LIN {X 0,Y 283.357,Z 583.66,A -85,B 0,C 180,E1 -18703.982,E2 -18703.982} C_VEL
LIN {X 0,Y 286.547,Z 569.765,A -85,B 0,C 180,E1 -18705.445,E2 -18705.445} C_VEL
LIN {X 0,Y 289.347,Z 555.188,A -85,B 0,C 180,E1 -18706.638,E2 -18706.638} C_VEL
LIN {X 0,Y 291.539,Z 540.137,A -85,B 0,C 180,E1 -18707.591,E2 -18707.591} C_VEL
LIN {X 0,Y 293.23,Z 524.888,A -85,B 0,C 180,E1 -18708.256,E2 -18708.256} C_VEL
LIN {X 0,Y 296.275,Z 478.654,A -85,B 0,C 180,E1 -18709.558,E2 -18709.558} C_VEL
LIN {X 0,Y 296.193,Z 472.889,A -85,B 0,C 180,E1 -18709.814,E2 -18709.814} C_VEL
LIN {X 0,Y 293.661,Z 454.463,A -85,B 0,C 180,E1 -18711.157,E2 -18711.157} C_VEL
LIN {X 0,Y 293.71,Z 448.696,A -85,B 0,C 180,E1 -18711.397,E2 -18711.397} C_VEL
LIN {X 0,Y 294.781,Z 433.314,A -85,B 0,C 180,E1 -18711.829,E2 -18711.829} C_VEL
LIN {X 0,Y 289.222,Z 422.71,A -85,B 0,C 180,E1 -18713.709,E2 -18713.709} C_VEL
LIN {X 0,Y 282.657,Z 411.761,A -85,B 0,C 180,E1 -18716.152,E2 -18716.152} C_VEL
LIN {X 0,Y 278.421,Z 405.383,A -85,B 0,C 180,E1 -18717.909,E2 -18717.909} C_VEL
LIN {X 0,Y 275.274,Z 400.843,A -85,B 0,C 180,E1 -18719.325,E2 -18719.325} C_VEL
LIN {X 0,Y 271.812,Z 395.922,A -85,B 0,C 180,E1 -18721.054,E2 -18721.054} C_VEL
LIN {X 0,Y 269.124,Z 392.173,A -85,B 0,C 180,E1 -18722.549,E2 -18722.549} C_VEL
LIN {X 0,Y 265.588,Z 388.374,A -85,B 0,C 180,E1 -18724.695,E2 -18724.695} C_VEL
LIN {X 0,Y 264.483,Z 386.612,A -85,B 0,C 180,E1 -18725.479,E2 -18725.479} C_VEL
LIN {X 0,Y 261.658,Z 384.021,A -85,B 0,C 180,E1 -18727.62,E2 -18727.62} C_VEL
LIN {X 0,Y 260.222,Z 381.079,A -85,B 0,C 180,E1 -18729.082,E2 -18729.082} C_VEL
LIN {X 0,Y 256.877,Z 379.067,A -85,B 0,C 180,E1 -18732.843,E2 -18732.843} C_VEL
LIN {X 0,Y 255.223,Z 375.845,A -85,B 0,C 180,E1 -18737.016,E2 -18737.016} C_VEL
LIN {X 0,Y 254.832,Z 376.279,A -85,B 0,C 180,E1 -18740.587,E2 -18740.587} C_VEL
LIN {X 0,Y 256.37,Z 378.534,A -85,B 0,C 180,E1 -18745.48,E2 -18745.48} C_VEL
LIN {X 0,Y 260.204,Z 384.567,A -85,B 0,C 180,E1 -18750.484,E2 -18750.484} C_VEL
LIN {X 0,Y 262.637,Z 387.768,A -85,B 0,C 180,E1 -18752.64,E2 -18752.64} C_VEL
LIN {X 0,Y 267.7,Z 395.205,A -85,B 0,C 180,E1 -18756.153,E2 -18756.153} C_VEL
LIN {X 0,Y 272.191,Z 402.334,A -85,B 0,C 180,E1 -18758.706,E2 -18758.706} C_VEL
LIN {X 0,Y 275.6,Z 407.992,A -85,B 0,C 180,E1 -18760.404,E2 -18760.404} C_VEL
LIN {X 0,Y 279.037,Z 414.108,A -85,B 0,C 180,E1 -18761.968,E2 -18761.968} C_VEL
LIN {X 0,Y 282.488,Z 420.477,A -85,B 0,C 180,E1 -18763.419,E2 -18763.419} C_VEL
LIN {X 0,Y 286.498,Z 428.65,A -85,B 0,C 180,E1 -18764.998,E2 -18764.998} C_VEL
LIN {X 0,Y 291.285,Z 439.57,A -85,B 0,C 180,E1 -18766.767,E2 -18766.767} C_VEL
LIN {X 0,Y 293.256,Z 444.964,A -85,B 0,C 180,E1 -18767.491,E2 -18767.491} C_VEL
LIN {X 0,Y 293.808,Z 453.087,A -85,B 0,C 180,E1 -18767.982,E2 -18767.982} C_VEL
LIN {X 0,Y 287.202,Z 546.54,A -85,B 0,C 180,E1 -18770.544,E2 -18770.544} C_VEL
LIN {X 0,Y 285.082,Z 562.821,A -85,B 0,C 180,E1 -18771.219,E2 -18771.219} C_VEL
LIN {X 0,Y 282.431,Z 577.753,A -85,B 0,C 180,E1 -18772.097,E2 -18772.097} C_VEL
LIN {X 0,Y 279.427,Z 591.001,A -85,B 0,C 180,E1 -18773.094,E2 -18773.094} C_VEL
LIN {X 0,Y 275.993,Z 604.177,A -85,B 0,C 180,E1 -18774.373,E2 -18774.373} C_VEL
LIN {X 0,Y 271.998,Z 617.923,A -85,B 0,C 180,E1 -18776.047,E2 -18776.047} C_VEL
LIN {X 0,Y 268.029,Z 630.286,A -85,B 0,C 180,E1 -18777.928,E2 -18777.928} C_VEL
LIN {X 0,Y 263.932,Z 641.731,A -85,B 0,C 180,E1 -18780.047,E2 -18780.047} C_VEL
LIN {X 0,Y 260.339,Z 651.436,A -85,B 0,C 180,E1 -18782.245,E2 -18782.245} C_VEL
LIN {X 0,Y 256.679,Z 661.36,A -85,B 0,C 180,E1 -18784.988,E2 -18784.988} C_VEL
LIN {X 0,Y 253.789,Z 669.171,A -85,B 0,C 180,E1 -18787.618,E2 -18787.618} C_VEL
LIN {X 0,Y 251.343,Z 675.969,A -85,B 0,C 180,E1 -18790.394,E2 -18790.394} C_VEL
LIN {X 0,Y 249.28,Z 682.278,A -85,B 0,C 180,E1 -18793.624,E2 -18793.624} C_VEL
LIN {X 0,Y 247.949,Z 687.204,A -85,B 0,C 180,E1 -18796.893,E2 -18796.893} C_VEL
LIN {X 0,Y 247.209,Z 690.852,A -85,B 0,C 180,E1 -18800.178,E2 -18800.178} C_VEL
LIN {X 0,Y 247.023,Z 693.292,A -85,B 0,C 180,E1 -18803.465,E2 -18803.465} C_VEL
LIN {X 0,Y 247.109,Z 694.554,A -85,B 0,C 180,E1 -18806.738,E2 -18806.738} C_VEL
LIN {X 0,Y 247.232,Z 694.628,A -85,B 0,C 180,E1 -18809.999,E2 -18809.999} C_VEL
LIN {X 0,Y 247.155,Z 693.435,A -85,B 0,C 180,E1 -18813.26,E2 -18813.26} C_VEL
LIN {X 0,Y 247.05,Z 690.958,A -85,B 0,C 180,E1 -18816.533,E2 -18816.533} C_VEL
LIN {X 0,Y 247.256,Z 687.184,A -85,B 0,C 180,E1 -18819.819,E2 -18819.819} C_VEL
LIN {X 0,Y 247.912,Z 682.014,A -85,B 0,C 180,E1 -18823.107,E2 -18823.107} C_VEL
LIN {X 0,Y 249.216,Z 675.046,A -85,B 0,C 180,E1 -18826.503,E2 -18826.503} C_VEL
LIN {X 0,Y 250.99,Z 666.908,A -85,B 0,C 180,E1 -18829.633,E2 -18829.633} C_VEL
LIN {X 0,Y 253.326,Z 657.918,A -85,B 0,C 180,E1 -18832.424,E2 -18832.424} C_VEL
LIN {X 0,Y 255.53,Z 648.604,A -85,B 0,C 180,E1 -18834.823,E2 -18834.823} C_VEL
LIN {X 0,Y 258.296,Z 637.846,A -85,B 0,C 180,E1 -18837.112,E2 -18837.112} C_VEL
LIN {X 0,Y 261.218,Z 626.014,A -85,B 0,C 180,E1 -18839.185,E2 -18839.185} C_VEL
LIN {X 0,Y 264.274,Z 613.144,A -85,B 0,C 180,E1 -18841.013,E2 -18841.013} C_VEL
LIN {X 0,Y 266.977,Z 600.152,A -85,B 0,C 180,E1 -18842.513,E2 -18842.513} C_VEL
LIN {X 0,Y 269.556,Z 585.357,A -85,B 0,C 180,E1 -18843.868,E2 -18843.868} C_VEL
LIN {X 0,Y 271.862,Z 570.467,A -85,B 0,C 180,E1 -18844.886,E2 -18844.886} C_VEL
LIN {X 0,Y 273.597,Z 555.142,A -85,B 0,C 180,E1 -18845.646,E2 -18845.646} C_VEL
LIN {X 0,Y 274.669,Z 537.879,A -85,B 0,C 180,E1 -18846.22,E2 -18846.22} C_VEL
LIN {X 0,Y 279.129,Z 449.321,A -85,B 0,C 180,E1 -18848.643,E2 -18848.643} C_VEL
LIN {X 0,Y 276.743,Z 432.647,A -85,B 0,C 180,E1 -18849.535,E2 -18849.535} C_VEL
LIN {X 0,Y 270.603,Z 418.098,A -85,B 0,C 180,E1 -18850.922,E2 -18850.922} C_VEL
LIN {X 0,Y 262.703,Z 401.029,A -85,B 0,C 180,E1 -18852.765,E2 -18852.765} C_VEL
LIN {X 0,Y 254.764,Z 385.449,A -85,B 0,C 180,E1 -18854.695,E2 -18854.695} C_VEL
LIN {X 0,Y 252.687,Z 381.306,A -85,B 0,C 180,E1 -18855.25,E2 -18855.25} C_VEL
LIN {X 0,Y 249.885,Z 372.112,A -85,B 0,C 180,E1 -18858.629,E2 -18858.629} C_VEL
LIN {X 0,Y 249.014,Z 369.094,A -85,B 0,C 180,E1 -18859.866,E2 -18859.866} C_VEL
LIN {X 0,Y 249.045,Z 369.092,A -85,B 0,C 180,E1 -18863.658,E2 -18863.658} C_VEL
LIN {X 0,Y 249.034,Z 369.085,A -85,B 0,C 180,E1 -18867.846,E2 -18867.846} C_VEL
LIN {X 0,Y 249.094,Z 369.082,A -85,B 0,C 180,E1 -18871.339,E2 -18871.339} C_VEL
LIN {X 0,Y 249.148,Z 369.073,A -85,B 0,C 180,E1 -18874.969,E2 -18874.969} C_VEL
LIN {X 0,Y 249.108,Z 369.08,A -85,B 0,C 180,E1 -18880.212,E2 -18880.212} C_VEL
LIN {X 0,Y 249.239,Z 369.065,A -85,B 0,C 180,E1 -18883.622,E2 -18883.622} C_VEL
LIN {X 0,Y 249.25,Z 369.033,A -85,B 0,C 180,E1 -18888.617,E2 -18888.617} C_VEL
LIN {X 0,Y 249.477,Z 369.026,A -85,B 0,C 180,E1 -18891.903,E2 -18891.903} C_VEL
LIN {X 0,Y 249.434,Z 369.031,A -85,B 0,C 180,E1 -18896.77,E2 -18896.77} C_VEL
LIN {X 0,Y 249.726,Z 368.993,A -85,B 0,C 180,E1 -18900.001,E2 -18900.001} C_VEL
LIN {X 0,Y 249.434,Z 369.038,A -85,B 0,C 180,E1 -18903.231,E2 -18903.231} C_VEL
LIN {X 0,Y 249.482,Z 369.017,A -85,B 0,C 180,E1 -18908.098,E2 -18908.098} C_VEL
LIN {X 0,Y 249.251,Z 369.062,A -85,B 0,C 180,E1 -18911.384,E2 -18911.384} C_VEL
LIN {X 0,Y 249.24,Z 369.043,A -85,B 0,C 180,E1 -18916.379,E2 -18916.379} C_VEL
LIN {X 0,Y 249.083,Z 369.081,A -85,B 0,C 180,E1 -18921.519,E2 -18921.519} C_VEL
LIN {X 0,Y 249.116,Z 369.057,A -85,B 0,C 180,E1 -18925.476,E2 -18925.476} C_VEL
LIN {X 0,Y 249.082,Z 369.082,A -85,B 0,C 180,E1 -18928.994,E2 -18928.994} C_VEL
LIN {X 0,Y 249.03,Z 369.085,A -85,B 0,C 180,E1 -18932.427,E2 -18932.427} C_VEL
LIN {X 0,Y 249.029,Z 369.076,A -85,B 0,C 180,E1 -18936.346,E2 -18936.346} C_VEL
LIN {X 0,Y 249.006,Z 369.092,A -85,B 0,C 180,E1 -18940.479,E2 -18940.479} C_VEL
LIN {X 0,Y 248.986,Z 369.084,A -85,B 0,C 180,E1 -18944.884,E2 -18944.884} C_VEL
LIN {X 0,Y 249.01,Z 369.092,A -85,B 0,C 180,E1 -18947.363,E2 -18947.363} C_VEL
LIN {X 0,Y 249.026,Z 369.075,A -85,B 0,C 180,E1 -18951.62,E2 -18951.62} C_VEL
LIN {X 0,Y 249.045,Z 369.087,A -85,B 0,C 180,E1 -18955.641,E2 -18955.641} C_VEL
LIN {X 0,Y 249.004,Z 369.087,A -85,B 0,C 180,E1 -18959.468,E2 -18959.468} C_VEL
LIN {X 0,Y 249.039,Z 369.082,A -85,B 0,C 180,E1 -18963.159,E2 -18963.159} C_VEL
LIN {X 0,Y 249.059,Z 369.087,A -85,B 0,C 180,E1 -18966.731,E2 -18966.731} C_VEL
LIN {X 0,Y 249.078,Z 369.076,A -85,B 0,C 180,E1 -18970.21,E2 -18970.21} C_VEL
LIN {X 0,Y 249.16,Z 369.069,A -85,B 0,C 180,E1 -18973.617,E2 -18973.617} C_VEL
LIN {X 0,Y 249.23,Z 369.06,A -85,B 0,C 180,E1 -18978.616,E2 -18978.616} C_VEL
LIN {X 0,Y 249.421,Z 369.036,A -85,B 0,C 180,E1 -18981.902,E2 -18981.902} C_VEL
LIN {X 0,Y 249.324,Z 369.179,A -85,B 0,C 180,E1 -18984.744,E2 -18984.744} C_VEL
LIN {X 0,Y 250.266,Z 371.871,A -85,B 0,C 180,E1 -18985.028,E2 -18985.028} C_VEL
LIN {X 0,Y 252.185,Z 374.531,A -85,B 0,C 180,E1 -18985.484,E2 -18985.484} C_VEL
LIN {X 0,Y 259.111,Z 385.318,A -85,B 0,C 180,E1 -18987.119,E2 -18987.119} C_VEL
LIN {X 0,Y 266.091,Z 397.678,A -85,B 0,C 180,E1 -18988.707,E2 -18988.707} C_VEL
LIN {X 0,Y 276.646,Z 417.563,A -85,B 0,C 180,E1 -18990.978,E2 -18990.978} C_VEL
LIN {X 0,Y 279.769,Z 424.265,A -85,B 0,C 180,E1 -18991.636,E2 -18991.636} C_VEL
LIN {X 0,Y 274.746,Z 521.539,A -85,B 0,C 180,E1 -18994.319,E2 -18994.319} C_VEL
LIN {X 0,Y 273.393,Z 537.132,A -85,B 0,C 180,E1 -18995.024,E2 -18995.024} C_VEL
LIN {X 0,Y 271.599,Z 552.606,A -85,B 0,C 180,E1 -18996.035,E2 -18996.035} C_VEL
LIN {X 0,Y 269.275,Z 567.725,A -85,B 0,C 180,E1 -18997.341,E2 -18997.341} C_VEL
LIN {X 0,Y 266.738,Z 581.835,A -85,B 0,C 180,E1 -18998.906,E2 -18998.906} C_VEL
LIN {X 0,Y 263.885,Z 595.218,A -85,B 0,C 180,E1 -19000.745,E2 -19000.745} C_VEL
LIN {X 0,Y 261.136,Z 607.122,A -85,B 0,C 180,E1 -19002.757,E2 -19002.757} C_VEL
LIN {X 0,Y 258.433,Z 617.973,A -85,B 0,C 180,E1 -19004.973,E2 -19004.973} C_VEL
LIN {X 0,Y 255.678,Z 628.541,A -85,B 0,C 180,E1 -19007.6,E2 -19007.6} C_VEL
LIN {X 0,Y 253.251,Z 637.668,A -85,B 0,C 180,E1 -19010.377,E2 -19010.377} C_VEL
LIN {X 0,Y 251.383,Z 644.892,A -85,B 0,C 180,E1 -19013.043,E2 -19013.043} C_VEL
LIN {X 0,Y 249.835,Z 651.011,A -85,B 0,C 180,E1 -19015.817,E2 -19015.817} C_VEL
LIN {X 0,Y 248.671,Z 656.327,A -85,B 0,C 180,E1 -19018.82,E2 -19018.82} C_VEL
LIN {X 0,Y 247.816,Z 660.314,A -85,B 0,C 180,E1 -19021.701,E2 -19021.701} C_VEL
LIN {X 0,Y 247.184,Z 663.356,A -85,B 0,C 180,E1 -19024.657,E2 -19024.657} C_VEL
LIN {X 0,Y 246.893,Z 665.098,A -85,B 0,C 180,E1 -19027.15,E2 -19027.15} C_VEL
LIN {X 0,Y 246.829,Z 666.221,A -85,B 0,C 180,E1 -19029.755,E2 -19029.755} C_VEL
LIN {X 0,Y 247.029,Z 666.573,A -85,B 0,C 180,E1 -19033.064,E2 -19033.064} C_VEL
LIN {X 0,Y 247.33,Z 666.182,A -85,B 0,C 180,E1 -19035.267,E2 -19035.267} C_VEL
LIN {X 0,Y 247.839,Z 665.251,A -85,B 0,C 180,E1 -19037.502,E2 -19037.502} C_VEL
LIN {X 0,Y 248.563,Z 663.696,A -85,B 0,C 180,E1 -19039.767,E2 -19039.767} C_VEL
LIN {X 0,Y 249.902,Z 660.558,A -85,B 0,C 180,E1 -19042.977,E2 -19042.977} C_VEL
LIN {X 0,Y 251.711,Z 656.351,A -85,B 0,C 180,E1 -19046.053,E2 -19046.053} C_VEL
LIN {X 0,Y 254.029,Z 650.936,A -85,B 0,C 180,E1 -19049.055,E2 -19049.055} C_VEL
LIN {X 0,Y 256.731,Z 644.578,A -85,B 0,C 180,E1 -19051.849,E2 -19051.849} C_VEL
LIN {X 0,Y 260.219,Z 636.264,A -85,B 0,C 180,E1 -19054.772,E2 -19054.772} C_VEL
LIN {X 0,Y 263.779,Z 627.473,A -85,B 0,C 180,E1 -19057.274,E2 -19057.274} C_VEL
LIN {X 0,Y 267.474,Z 617.456,A -85,B 0,C 180,E1 -19059.625,E2 -19059.625} C_VEL
LIN {X 0,Y 271.215,Z 606.687,A -85,B 0,C 180,E1 -19061.687,E2 -19061.687} C_VEL
LIN {X 0,Y 274.829,Z 595.249,A -85,B 0,C 180,E1 -19063.488,E2 -19063.488} C_VEL
LIN {X 0,Y 278.429,Z 582.521,A -85,B 0,C 180,E1 -19065.12,E2 -19065.12} C_VEL
LIN {X 0,Y 281.53,Z 569.386,A -85,B 0,C 180,E1 -19066.501,E2 -19066.501} C_VEL
LIN {X 0,Y 284.323,Z 555.435,A -85,B 0,C 180,E1 -19067.644,E2 -19067.644} C_VEL
LIN {X 0,Y 286.501,Z 541.074,A -85,B 0,C 180,E1 -19068.561,E2 -19068.561} C_VEL
LIN {X 0,Y 288.235,Z 525.976,A -85,B 0,C 180,E1 -19069.24,E2 -19069.24} C_VEL
LIN {X 0,Y 291.553,Z 478.481,A -85,B 0,C 180,E1 -19070.59,E2 -19070.59} C_VEL
LIN {X 0,Y 293.71,Z 448.696,A -85,B 0,C 180,E1 -19071.397,E2 -19071.397} C_VEL
LIN {X 0,Y 293.59,Z 444.895,A -85,B 0,C 180,E1 -19071.596,E2 -19071.596} C_VEL
LIN {X 0,Y 292.386,Z 440.371,A -85,B 0,C 180,E1 -19072.09,E2 -19072.09} C_VEL
LIN {X 0,Y 289.941,Z 435.432,A -85,B 0,C 180,E1 -19072.925,E2 -19072.925} C_VEL
LIN {X 0,Y 287.813,Z 431.718,A -85,B 0,C 180,E1 -19073.65,E2 -19073.65} C_VEL
LIN {X 0,Y 282.661,Z 422.453,A -85,B 0,C 180,E1 -19075.585,E2 -19075.585} C_VEL
LIN {X 0,Y 277.736,Z 414.214,A -85,B 0,C 180,E1 -19077.626,E2 -19077.626} C_VEL
LIN {X 0,Y 271.268,Z 404.805,A -85,B 0,C 180,E1 -19080.664,E2 -19080.664} C_VEL
LIN {X 0,Y 269.595,Z 402.252,A -85,B 0,C 180,E1 -19081.563,E2 -19081.563} C_VEL
LIN {X 0,Y 266.623,Z 398.146,A -85,B 0,C 180,E1 -19083.305,E2 -19083.305} C_VEL
LIN {X 0,Y 263.648,Z 394.765,A -85,B 0,C 180,E1 -19085.209,E2 -19085.209} C_VEL
LIN {X 0,Y 262.663,Z 393.245,A -85,B 0,C 180,E1 -19085.951,E2 -19085.951} C_VEL
LIN {X 0,Y 259.912,Z 390.436,A -85,B 0,C 180,E1 -19088.174,E2 -19088.174} C_VEL
LIN {X 0,Y 258.564,Z 387.874,A -85,B 0,C 180,E1 -19089.583,E2 -19089.583} C_VEL
LIN {X 0,Y 255.368,Z 385.663,A -85,B 0,C 180,E1 -19093.528,E2 -19093.528} C_VEL
LIN {X 0,Y 254.133,Z 382.889,A -85,B 0,C 180,E1 -19097.092,E2 -19097.092} C_VEL
LIN {X 0,Y 253.747,Z 383.264,A -85,B 0,C 180,E1 -19100.403,E2 -19100.403} C_VEL
LIN {X 0,Y 255.238,Z 385.561,A -85,B 0,C 180,E1 -19105.397,E2 -19105.397} C_VEL
LIN {X 0,Y 258.718,Z 391.354,A -85,B 0,C 180,E1 -19110.142,E2 -19110.142} C_VEL
LIN {X 0,Y 260.948,Z 394.357,A -85,B 0,C 180,E1 -19112.188,E2 -19112.188} C_VEL
LIN {X 0,Y 265.509,Z 401.376,A -85,B 0,C 180,E1 -19115.551,E2 -19115.551} C_VEL
LIN {X 0,Y 269.578,Z 408.07,A -85,B 0,C 180,E1 -19118.001,E2 -19118.001} C_VEL
LIN {X 0,Y 273.017,Z 414.016,A -85,B 0,C 180,E1 -19119.814,E2 -19119.814} C_VEL
LIN {X 0,Y 275.844,Z 419.193,A -85,B 0,C 180,E1 -19121.173,E2 -19121.173} C_VEL
LIN {X 0,Y 280.027,Z 427.177,A -85,B 0,C 180,E1 -19123.026,E2 -19123.026} C_VEL
LIN {X 0,Y 284.416,Z 436.813,A -85,B 0,C 180,E1 -19124.823,E2 -19124.823} C_VEL
LIN {X 0,Y 288.38,Z 446.669,A -85,B 0,C 180,E1 -19126.365,E2 -19126.365} C_VEL
LIN {X 0,Y 288.92,Z 448.494,A -85,B 0,C 180,E1 -19126.586,E2 -19126.586} C_VEL
LIN {X 0,Y 289.262,Z 453.9,A -85,B 0,C 180,E1 -19126.92,E2 -19126.92} C_VEL
LIN {X 0,Y 282.349,Z 546.363,A -85,B 0,C 180,E1 -19129.495,E2 -19129.495} C_VEL
LIN {X 0,Y 280.173,Z 562.533,A -85,B 0,C 180,E1 -19130.175,E2 -19130.175} C_VEL
LIN {X 0,Y 277.653,Z 576.328,A -85,B 0,C 180,E1 -19130.976,E2 -19130.976} C_VEL
LIN {X 0,Y 274.318,Z 590.651,A -85,B 0,C 180,E1 -19132.056,E2 -19132.056} C_VEL
LIN {X 0,Y 270.342,Z 605.304,A -85,B 0,C 180,E1 -19133.51,E2 -19133.51} C_VEL
LIN {X 0,Y 266.188,Z 618.701,A -85,B 0,C 180,E1 -19135.201,E2 -19135.201} C_VEL
LIN {X 0,Y 262.061,Z 630.826,A -85,B 0,C 180,E1 -19137.106,E2 -19137.106} C_VEL
LIN {X 0,Y 257.817,Z 642.124,A -85,B 0,C 180,E1 -19139.261,E2 -19139.261} C_VEL
LIN {X 0,Y 253.476,Z 653.199,A -85,B 0,C 180,E1 -19141.877,E2 -19141.877} C_VEL
LIN {X 0,Y 250.028,Z 661.958,A -85,B 0,C 180,E1 -19144.443,E2 -19144.443} C_VEL
LIN {X 0,Y 247.197,Z 669.166,A -85,B 0,C 180,E1 -19146.987,E2 -19146.987} C_VEL
LIN {X 0,Y 244.593,Z 675.876,A -85,B 0,C 180,E1 -19149.83,E2 -19149.83} C_VEL
LIN {X 0,Y 242.422,Z 682.119,A -85,B 0,C 180,E1 -19153.147,E2 -19153.147} C_VEL
LIN {X 0,Y 240.967,Z 686.994,A -85,B 0,C 180,E1 -19156.506,E2 -19156.506} C_VEL
LIN {X 0,Y 240.139,Z 690.566,A -85,B 0,C 180,E1 -19159.886,E2 -19159.886} C_VEL
LIN {X 0,Y 239.941,Z 692.948,A -85,B 0,C 180,E1 -19163.271,E2 -19163.271} C_VEL
LIN {X 0,Y 240.018,Z 694.15,A -85,B 0,C 180,E1 -19166.642,E2 -19166.642} C_VEL
LIN {X 0,Y 240.152,Z 694.166,A -85,B 0,C 180,E1 -19169.999,E2 -19169.999} C_VEL
LIN {X 0,Y 240.061,Z 692.937,A -85,B 0,C 180,E1 -19173.356,E2 -19173.356} C_VEL
LIN {X 0,Y 239.965,Z 690.401,A -85,B 0,C 180,E1 -19176.727,E2 -19176.727} C_VEL
LIN {X 0,Y 240.197,Z 686.556,A -85,B 0,C 180,E1 -19180.11,E2 -19180.11} C_VEL
LIN {X 0,Y 240.917,Z 681.31,A -85,B 0,C 180,E1 -19183.495,E2 -19183.495} C_VEL
LIN {X 0,Y 242.259,Z 674.532,A -85,B 0,C 180,E1 -19186.863,E2 -19186.863} C_VEL
LIN {X 0,Y 243.917,Z 667.174,A -85,B 0,C 180,E1 -19189.788,E2 -19189.788} C_VEL
LIN {X 0,Y 246.293,Z 658.32,A -85,B 0,C 180,E1 -19192.657,E2 -19192.657} C_VEL
LIN {X 0,Y 248.949,Z 647.763,A -85,B 0,C 180,E1 -19195.454,E2 -19195.454} C_VEL
LIN {X 0,Y 251.88,Z 636.593,A -85,B 0,C 180,E1 -19197.862,E2 -19197.862} C_VEL
LIN {X 0,Y 254.953,Z 624.595,A -85,B 0,C 180,E1 -19199.975,E2 -19199.975} C_VEL
LIN {X 0,Y 258.076,Z 611.495,A -85,B 0,C 180,E1 -19201.844,E2 -19201.844} C_VEL
LIN {X 0,Y 261.12,Z 597.349,A -85,B 0,C 180,E1 -19203.451,E2 -19203.451} C_VEL
LIN {X 0,Y 263.641,Z 583.048,A -85,B 0,C 180,E1 -19204.736,E2 -19204.736} C_VEL
LIN {X 0,Y 265.994,Z 567.521,A -85,B 0,C 180,E1 -19205.772,E2 -19205.772} C_VEL
LIN {X 0,Y 267.644,Z 552.107,A -85,B 0,C 180,E1 -19206.506,E2 -19206.506} C_VEL
LIN {X 0,Y 269.042,Z 528.766,A -85,B 0,C 180,E1 -19207.22,E2 -19207.22} C_VEL
LIN {X 0,Y 273.126,Z 450.076,A -85,B 0,C 180,E1 -19209.419,E2 -19209.419} C_VEL
LIN {X 0,Y 271.018,Z 435.37,A -85,B 0,C 180,E1 -19210.238,E2 -19210.238} C_VEL
LIN {X 0,Y 263.905,Z 418.352,A -85,B 0,C 180,E1 -19211.925,E2 -19211.925} C_VEL
LIN {X 0,Y 254.711,Z 398.936,A -85,B 0,C 180,E1 -19214.161,E2 -19214.161} C_VEL
LIN {X 0,Y 247.112,Z 384.535,A -85,B 0,C 180,E1 -19216.104,E2 -19216.104} C_VEL
LIN {X 0,Y 245.235,Z 380.665,A -85,B 0,C 180,E1 -19216.686,E2 -19216.686} C_VEL
LIN {X 0,Y 241.99,Z 369.959,A -85,B 0,C 180,E1 -19220.853,E2 -19220.853} C_VEL
LIN {X 0,Y 241.985,Z 369.974,A -85,B 0,C 180,E1 -19224.489,E2 -19224.489} C_VEL
LIN {X 0,Y 241.972,Z 369.97,A -85,B 0,C 180,E1 -19228.48,E2 -19228.48} C_VEL
LIN {X 0,Y 242.006,Z 369.966,A -85,B 0,C 180,E1 -19232.313,E2 -19232.313} C_VEL
LIN {X 0,Y 242.054,Z 369.958,A -85,B 0,C 180,E1 -19236.016,E2 -19236.016} C_VEL
LIN {X 0,Y 242.035,Z 369.962,A -85,B 0,C 180,E1 -19239.608,E2 -19239.608} C_VEL
LIN {X 0,Y 242.16,Z 369.947,A -85,B 0,C 180,E1 -19243.279,E2 -19243.279} C_VEL
LIN {X 0,Y 242.184,Z 369.913,A -85,B 0,C 180,E1 -19248.28,E2 -19248.28} C_VEL
LIN {X 0,Y 242.424,Z 369.9,A -85,B 0,C 180,E1 -19251.666,E2 -19251.666} C_VEL
LIN {X 0,Y 242.257,Z 369.934,A -85,B 0,C 180,E1 -19255.008,E2 -19255.008} C_VEL
LIN {X 0,Y 242.634,Z 369.868,A -85,B 0,C 180,E1 -19258.341,E2 -19258.341} C_VEL
LIN {X 0,Y 242.635,Z 369.884,A -85,B 0,C 180,E1 -19261.66,E2 -19261.66} C_VEL
LIN {X 0,Y 242.429,Z 369.893,A -85,B 0,C 180,E1 -19266.709,E2 -19266.709} C_VEL
LIN {X 0,Y 242.344,Z 369.917,A -85,B 0,C 180,E1 -19270.021,E2 -19270.021} C_VEL
LIN {X 0,Y 242.165,Z 369.928,A -85,B 0,C 180,E1 -19275.142,E2 -19275.142} C_VEL
LIN {X 0,Y 242.071,Z 369.947,A -85,B 0,C 180,E1 -19278.625,E2 -19278.625} C_VEL
LIN {X 0,Y 242.005,Z 369.964,A -85,B 0,C 180,E1 -19282.181,E2 -19282.181} C_VEL
LIN {X 0,Y 242.065,Z 369.933,A -85,B 0,C 180,E1 -19285.839,E2 -19285.839} C_VEL
LIN {X 0,Y 242.029,Z 369.96,A -85,B 0,C 180,E1 -19289.581,E2 -19289.581} C_VEL
LIN {X 0,Y 241.98,Z 369.956,A -85,B 0,C 180,E1 -19293.494,E2 -19293.494} C_VEL
LIN {X 0,Y 241.986,Z 369.962,A -85,B 0,C 180,E1 -19297.583,E2 -19297.583} C_VEL
LIN {X 0,Y 241.933,Z 369.965,A -85,B 0,C 180,E1 -19301.924,E2 -19301.924} C_VEL
LIN {X 0,Y 241.926,Z 369.974,A -85,B 0,C 180,E1 -19306.575,E2 -19306.575} C_VEL
LIN {X 0,Y 241.957,Z 369.959,A -85,B 0,C 180,E1 -19310.282,E2 -19310.282} C_VEL
LIN {X 0,Y 241.989,Z 369.969,A -85,B 0,C 180,E1 -19314.49,E2 -19314.49} C_VEL
LIN {X 0,Y 241.954,Z 369.959,A -85,B 0,C 180,E1 -19318.478,E2 -19318.478} C_VEL
LIN {X 0,Y 241.972,Z 369.968,A -85,B 0,C 180,E1 -19322.309,E2 -19322.309} C_VEL
LIN {X 0,Y 242.029,Z 369.958,A -85,B 0,C 180,E1 -19326.014,E2 -19326.014} C_VEL
LIN {X 0,Y 242.018,Z 369.953,A -85,B 0,C 180,E1 -19329.607,E2 -19329.607} C_VEL
LIN {X 0,Y 242.108,Z 369.948,A -85,B 0,C 180,E1 -19333.325,E2 -19333.325} C_VEL
LIN {X 0,Y 242.162,Z 369.939,A -85,B 0,C 180,E1 -19338.279,E2 -19338.279} C_VEL
LIN {X 0,Y 242.375,Z 369.913,A -85,B 0,C 180,E1 -19341.665,E2 -19341.665} C_VEL
LIN {X 0,Y 242.394,Z 369.918,A -85,B 0,C 180,E1 -19343.435,E2 -19343.435} C_VEL
LIN {X 0,Y 243.474,Z 372.961,A -85,B 0,C 180,E1 -19343.802,E2 -19343.802} C_VEL
LIN {X 0,Y 245.055,Z 375.31,A -85,B 0,C 180,E1 -19344.207,E2 -19344.207} C_VEL
LIN {X 0,Y 254.562,Z 390.102,A -85,B 0,C 180,E1 -19346.535,E2 -19346.535} C_VEL
LIN {X 0,Y 261.4,Z 402.403,A -85,B 0,C 180,E1 -19348.153,E2 -19348.153} C_VEL
LIN {X 0,Y 271.387,Z 421.335,A -85,B 0,C 180,E1 -19350.363,E2 -19350.363} C_VEL
LIN {X 0,Y 273.748,Z 426.672,A -85,B 0,C 180,E1 -19350.889,E2 -19350.889} C_VEL
LIN {X 0,Y 268.582,Z 522.332,A -85,B 0,C 180,E1 -19353.583,E2 -19353.583} C_VEL
LIN {X 0,Y 267.21,Z 537.779,A -85,B 0,C 180,E1 -19354.303,E2 -19354.303} C_VEL
LIN {X 0,Y 265.385,Z 553.005,A -85,B 0,C 180,E1 -19355.319,E2 -19355.319} C_VEL
LIN {X 0,Y 263.047,Z 567.686,A -85,B 0,C 180,E1 -19356.603,E2 -19356.603} C_VEL
LIN {X 0,Y 260.519,Z 581.439,A -85,B 0,C 180,E1 -19358.143,E2 -19358.143} C_VEL
LIN {X 0,Y 257.633,Z 594.717,A -85,B 0,C 180,E1 -19359.982,E2 -19359.982} C_VEL
LIN {X 0,Y 254.863,Z 606.282,A -85,B 0,C 180,E1 -19361.937,E2 -19361.937} C_VEL
LIN {X 0,Y 252.003,Z 617.513,A -85,B 0,C 180,E1 -19364.244,E2 -19364.244} C_VEL
LIN {X 0,Y 249.11,Z 628.183,A -85,B 0,C 180,E1 -19366.917,E2 -19366.917} C_VEL
LIN {X 0,Y 246.515,Z 637.583,A -85,B 0,C 180,E1 -19369.81,E2 -19369.81} C_VEL
LIN {X 0,Y 244.275,Z 645.879,A -85,B 0,C 180,E1 -19372.974,E2 -19372.974} C_VEL
LIN {X 0,Y 242.609,Z 652.448,A -85,B 0,C 180,E1 -19376.099,E2 -19376.099} C_VEL
LIN {X 0,Y 241.452,Z 657.514,A -85,B 0,C 180,E1 -19379.164,E2 -19379.164} C_VEL
LIN {X 0,Y 240.613,Z 661.264,A -85,B 0,C 180,E1 -19382.106,E2 -19382.106} C_VEL
LIN {X 0,Y 239.903,Z 664.66,A -85,B 0,C 180,E1 -19385.868,E2 -19385.868} C_VEL
LIN {X 0,Y 239.749,Z 665.917,A -85,B 0,C 180,E1 -19387.996,E2 -19387.996} C_VEL
LIN {X 0,Y 239.753,Z 666.78,A -85,B 0,C 180,E1 -19390.345,E2 -19390.345} C_VEL
LIN {X 0,Y 239.923,Z 667.017,A -85,B 0,C 180,E1 -19392.918,E2 -19392.918} C_VEL
LIN {X 0,Y 240.276,Z 666.651,A -85,B 0,C 180,E1 -19395.412,E2 -19395.412} C_VEL
LIN {X 0,Y 240.846,Z 665.711,A -85,B 0,C 180,E1 -19397.843,E2 -19397.843} C_VEL
LIN {X 0,Y 242.198,Z 663.013,A -85,B 0,C 180,E1 -19401.581,E2 -19401.581} C_VEL
LIN {X 0,Y 243.836,Z 659.445,A -85,B 0,C 180,E1 -19404.798,E2 -19404.798} C_VEL
LIN {X 0,Y 245.991,Z 654.689,A -85,B 0,C 180,E1 -19407.96,E2 -19407.96} C_VEL
LIN {X 0,Y 249.005,Z 648.088,A -85,B 0,C 180,E1 -19411.326,E2 -19411.326} C_VEL
LIN {X 0,Y 252.592,Z 640.15,A -85,B 0,C 180,E1 -19414.468,E2 -19414.468} C_VEL
LIN {X 0,Y 256.141,Z 631.986,A -85,B 0,C 180,E1 -19417.05,E2 -19417.05} C_VEL
LIN {X 0,Y 260.209,Z 621.838,A -85,B 0,C 180,E1 -19419.674,E2 -19419.674} C_VEL
LIN {X 0,Y 264.363,Z 610.756,A -85,B 0,C 180,E1 -19421.988,E2 -19421.988} C_VEL
LIN {X 0,Y 268.406,Z 598.99,A -85,B 0,C 180,E1 -19423.981,E2 -19423.981} C_VEL
LIN {X 0,Y 271.961,Z 587.339,A -85,B 0,C 180,E1 -19425.597,E2 -19425.597} C_VEL
LIN {X 0,Y 275.705,Z 572.943,A -85,B 0,C 180,E1 -19427.213,E2 -19427.213} C_VEL
LIN {X 0,Y 278.796,Z 558.737,A -85,B 0,C 180,E1 -19428.45,E2 -19428.45} C_VEL
LIN {X 0,Y 281.264,Z 543.966,A -85,B 0,C 180,E1 -19429.452,E2 -19429.452} C_VEL
LIN {X 0,Y 283.126,Z 529.014,A -85,B 0,C 180,E1 -19430.19,E2 -19430.19} C_VEL
LIN {X 0,Y 284.855,Z 507.429,A -85,B 0,C 180,E1 -19430.871,E2 -19430.871} C_VEL
LIN {X 0,Y 290.118,Z 436.331,A -85,B 0,C 180,E1 -19432.838,E2 -19432.838} C_VEL
LIN {X 0,Y 287.813,Z 431.718,A -85,B 0,C 180,E1 -19433.65,E2 -19433.65} C_VEL
LIN {X 0,Y 285.384,Z 428.368,A -85,B 0,C 180,E1 -19434.492,E2 -19434.492} C_VEL
LIN {X 0,Y 280.656,Z 424.632,A -85,B 0,C 180,E1 -19436.091,E2 -19436.091} C_VEL
LIN {X 0,Y 276.925,Z 421.974,A -85,B 0,C 180,E1 -19437.45,E2 -19437.45} C_VEL
LIN {X 0,Y 274.5,Z 419.37,A -85,B 0,C 180,E1 -19438.45,E2 -19438.45} C_VEL
LIN {X 0,Y 273.809,Z 418.287,A -85,B 0,C 180,E1 -19438.769,E2 -19438.769} C_VEL
LIN {X 0,Y 267.458,Z 408.611,A -85,B 0,C 180,E1 -19442.07,E2 -19442.07} C_VEL
LIN {X 0,Y 264.525,Z 404.517,A -85,B 0,C 180,E1 -19443.861,E2 -19443.861} C_VEL
LIN {X 0,Y 261.632,Z 400.962,A -85,B 0,C 180,E1 -19445.835,E2 -19445.835} C_VEL
LIN {X 0,Y 260.794,Z 399.816,A -85,B 0,C 180,E1 -19446.479,E2 -19446.479} C_VEL
LIN {X 0,Y 258.132,Z 396.797,A -85,B 0,C 180,E1 -19448.789,E2 -19448.789} C_VEL
LIN {X 0,Y 257.203,Z 394.804,A -85,B 0,C 180,E1 -19449.833,E2 -19449.833} C_VEL
LIN {X 0,Y 254.128,Z 392.549,A -85,B 0,C 180,E1 -19453.799,E2 -19453.799} C_VEL
LIN {X 0,Y 253.01,Z 389.805,A -85,B 0,C 180,E1 -19457.377,E2 -19457.377} C_VEL
LIN {X 0,Y 252.722,Z 390.452,A -85,B 0,C 180,E1 -19460.83,E2 -19460.83} C_VEL
LIN {X 0,Y 254.06,Z 392.523,A -85,B 0,C 180,E1 -19465.227,E2 -19465.227} C_VEL
LIN {X 0,Y 257.509,Z 398.495,A -85,B 0,C 180,E1 -19470.063,E2 -19470.063} C_VEL
LIN {X 0,Y 259.275,Z 400.981,A -85,B 0,C 180,E1 -19471.734,E2 -19471.734} C_VEL
LIN {X 0,Y 263.459,Z 407.727,A -85,B 0,C 180,E1 -19475.013,E2 -19475.013} C_VEL
LIN {X 0,Y 267.312,Z 414.333,A -85,B 0,C 180,E1 -19477.455,E2 -19477.455} C_VEL
LIN {X 0,Y 270.399,Z 419.842,A -85,B 0,C 180,E1 -19479.158,E2 -19479.158} C_VEL
LIN {X 0,Y 273.533,Z 425.888,A -85,B 0,C 180,E1 -19480.758,E2 -19480.758} C_VEL
LIN {X 0,Y 277.061,Z 432.96,A -85,B 0,C 180,E1 -19482.389,E2 -19482.389} C_VEL
LIN {X 0,Y 280.694,Z 441.175,A -85,B 0,C 180,E1 -19483.971,E2 -19483.971} C_VEL
LIN {X 0,Y 284.505,Z 451.056,A -85,B 0,C 180,E1 -19485.561,E2 -19485.561} C_VEL
LIN {X 0,Y 284.758,Z 455.497,A -85,B 0,C 180,E1 -19485.846,E2 -19485.846} C_VEL
LIN {X 0,Y 277.751,Z 545.662,A -85,B 0,C 180,E1 -19488.378,E2 -19488.378} C_VEL
LIN {X 0,Y 275.497,Z 561.794,A -85,B 0,C 180,E1 -19489.057,E2 -19489.057} C_VEL
LIN {X 0,Y 272.743,Z 576.131,A -85,B 0,C 180,E1 -19489.894,E2 -19489.894} C_VEL
LIN {X 0,Y 269.301,Z 590.327,A -85,B 0,C 180,E1 -19490.979,E2 -19490.979} C_VEL
LIN {X 0,Y 265.155,Z 604.933,A -85,B 0,C 180,E1 -19492.437,E2 -19492.437} C_VEL
LIN {X 0,Y 260.843,Z 618.315,A -85,B 0,C 180,E1 -19494.143,E2 -19494.143} C_VEL
LIN {X 0,Y 256.535,Z 630.441,A -85,B 0,C 180,E1 -19496.068,E2 -19496.068} C_VEL
LIN {X 0,Y 251.76,Z 642.532,A -85,B 0,C 180,E1 -19498.438,E2 -19498.438} C_VEL
LIN {X 0,Y 247.23,Z 653.413,A -85,B 0,C 180,E1 -19501.101,E2 -19501.101} C_VEL
LIN {X 0,Y 243.507,Z 662.335,A -85,B 0,C 180,E1 -19503.79,E2 -19503.79} C_VEL
LIN {X 0,Y 240.202,Z 670.252,A -85,B 0,C 180,E1 -19506.734,E2 -19506.734} C_VEL
LIN {X 0,Y 237.22,Z 677.483,A -85,B 0,C 180,E1 -19510.079,E2 -19510.079} C_VEL
LIN {X 0,Y 235.08,Z 683.346,A -85,B 0,C 180,E1 -19513.552,E2 -19513.552} C_VEL
LIN {X 0,Y 234.001,Z 686.773,A -85,B 0,C 180,E1 -19516.097,E2 -19516.097} C_VEL
LIN {X 0,Y 233.084,Z 690.3,A -85,B 0,C 180,E1 -19519.576,E2 -19519.576} C_VEL
LIN {X 0,Y 232.86,Z 692.608,A -85,B 0,C 180,E1 -19523.065,E2 -19523.065} C_VEL
LIN {X 0,Y 232.93,Z 693.749,A -85,B 0,C 180,E1 -19526.54,E2 -19526.54} C_VEL
LIN {X 0,Y 233.073,Z 693.704,A -85,B 0,C 180,E1 -19529.999,E2 -19529.999} C_VEL
LIN {X 0,Y 232.972,Z 692.421,A -85,B 0,C 180,E1 -19533.458,E2 -19533.458} C_VEL
LIN {X 0,Y 232.951,Z 691.146,A -85,B 0,C 180,E1 -19535.387,E2 -19535.387} C_VEL
LIN {X 0,Y 232.982,Z 688.053,A -85,B 0,C 180,E1 -19538.674,E2 -19538.674} C_VEL
LIN {X 0,Y 233.43,Z 683.442,A -85,B 0,C 180,E1 -19542.166,E2 -19542.166} C_VEL
LIN {X 0,Y 234.554,Z 677.37,A -85,B 0,C 180,E1 -19545.644,E2 -19545.644} C_VEL
LIN {X 0,Y 236.315,Z 669.669,A -85,B 0,C 180,E1 -19549.094,E2 -19549.094} C_VEL
LIN {X 0,Y 238.515,Z 661.385,A -85,B 0,C 180,E1 -19552.066,E2 -19552.066} C_VEL
LIN {X 0,Y 241.156,Z 651.552,A -85,B 0,C 180,E1 -19554.95,E2 -19554.95} C_VEL
LIN {X 0,Y 243.991,Z 641.16,A -85,B 0,C 180,E1 -19557.442,E2 -19557.442} C_VEL
LIN {X 0,Y 247.001,Z 630.087,A -85,B 0,C 180,E1 -19559.628,E2 -19559.628} C_VEL
LIN {X 0,Y 250.061,Z 618.161,A -85,B 0,C 180,E1 -19561.564,E2 -19561.564} C_VEL
LIN {X 0,Y 253.099,Z 605.317,A -85,B 0,C 180,E1 -19563.257,E2 -19563.257} C_VEL
LIN {X 0,Y 255.899,Z 591.101,A -85,B 0,C 180,E1 -19564.767,E2 -19564.767} C_VEL
LIN {X 0,Y 258.529,Z 575.806,A -85,B 0,C 180,E1 -19566.005,E2 -19566.005} C_VEL
LIN {X 0,Y 260.547,Z 561.064,A -85,B 0,C 180,E1 -19566.881,E2 -19566.881} C_VEL
LIN {X 0,Y 262.004,Z 546.383,A -85,B 0,C 180,E1 -19567.485,E2 -19567.485} C_VEL
LIN {X 0,Y 267.205,Z 451.465,A -85,B 0,C 180,E1 -19570.206,E2 -19570.206} C_VEL
LIN {X 0,Y 265.387,Z 438.14,A -85,B 0,C 180,E1 -19570.963,E2 -19570.963} C_VEL
LIN {X 0,Y 259.249,Z 423.406,A -85,B 0,C 180,E1 -19572.454,E2 -19572.454} C_VEL
LIN {X 0,Y 250.263,Z 403.939,A -85,B 0,C 180,E1 -19574.731,E2 -19574.731} C_VEL
LIN {X 0,Y 242.038,Z 388.298,A -85,B 0,C 180,E1 -19576.901,E2 -19576.901} C_VEL
LIN {X 0,Y 237.844,Z 380.27,A -85,B 0,C 180,E1 -19578.126,E2 -19578.126} C_VEL
LIN {X 0,Y 234.952,Z 370.832,A -85,B 0,C 180,E1 -19582.043,E2 -19582.043} C_VEL
LIN {X 0,Y 234.939,Z 370.833,A -85,B 0,C 180,E1 -19586.885,E2 -19586.885} C_VEL
LIN {X 0,Y 234.949,Z 370.844,A -85,B 0,C 180,E1 -19591.406,E2 -19591.406} C_VEL
LIN {X 0,Y 234.984,Z 370.839,A -85,B 0,C 180,E1 -19595.247,E2 -19595.247} C_VEL
LIN {X 0,Y 235.008,Z 370.836,A -85,B 0,C 180,E1 -19598.97,E2 -19598.97} C_VEL
LIN {X 0,Y 235.093,Z 370.825,A -85,B 0,C 180,E1 -19603.06,E2 -19603.06} C_VEL
LIN {X 0,Y 235.116,Z 370.795,A -85,B 0,C 180,E1 -19607.923,E2 -19607.923} C_VEL
LIN {X 0,Y 235.373,Z 370.773,A -85,B 0,C 180,E1 -19611.415,E2 -19611.415} C_VEL
LIN {X 0,Y 235.4,Z 370.785,A -85,B 0,C 180,E1 -19613.142,E2 -19613.142} C_VEL
LIN {X 0,Y 235.594,Z 370.744,A -85,B 0,C 180,E1 -19618.291,E2 -19618.291} C_VEL
LIN {X 0,Y 235.594,Z 370.761,A -85,B 0,C 180,E1 -19621.71,E2 -19621.71} C_VEL
LIN {X 0,Y 235.404,Z 370.766,A -85,B 0,C 180,E1 -19626.859,E2 -19626.859} C_VEL
LIN {X 0,Y 235.252,Z 370.802,A -85,B 0,C 180,E1 -19630.327,E2 -19630.327} C_VEL
LIN {X 0,Y 235.112,Z 370.804,A -85,B 0,C 180,E1 -19635.607,E2 -19635.607} C_VEL
LIN {X 0,Y 235.006,Z 370.832,A -85,B 0,C 180,E1 -19639.206,E2 -19639.206} C_VEL
LIN {X 0,Y 234.951,Z 370.838,A -85,B 0,C 180,E1 -19642.885,E2 -19642.885} C_VEL
LIN {X 0,Y 234.968,Z 370.819,A -85,B 0,C 180,E1 -19646.658,E2 -19646.658} C_VEL
LIN {X 0,Y 234.931,Z 370.848,A -85,B 0,C 180,E1 -19650.569,E2 -19650.569} C_VEL
LIN {X 0,Y 234.926,Z 370.826,A -85,B 0,C 180,E1 -19654.64,E2 -19654.64} C_VEL
LIN {X 0,Y 234.941,Z 370.846,A -85,B 0,C 180,E1 -19658.945,E2 -19658.945} C_VEL
LIN {X 0,Y 234.878,Z 370.832,A -85,B 0,C 180,E1 -19663.489,E2 -19663.489} C_VEL
LIN {X 0,Y 234.878,Z 370.851,A -85,B 0,C 180,E1 -19666.513,E2 -19666.513} C_VEL
LIN {X 0,Y 234.918,Z 370.831,A -85,B 0,C 180,E1 -19671.08,E2 -19671.08} C_VEL
LIN {X 0,Y 234.931,Z 370.846,A -85,B 0,C 180,E1 -19675.363,E2 -19675.363} C_VEL
LIN {X 0,Y 234.9,Z 370.843,A -85,B 0,C 180,E1 -19679.429,E2 -19679.429} C_VEL
LIN {X 0,Y 234.971,Z 370.831,A -85,B 0,C 180,E1 -19683.808,E2 -19683.808} C_VEL
LIN {X 0,Y 234.971,Z 370.831,A -85,B 0,C 180,E1 -19688.967,E2 -19688.967} C_VEL
LIN {X 0,Y 235.052,Z 370.828,A -85,B 0,C 180,E1 -19693.098,E2 -19693.098} C_VEL
LIN {X 0,Y 235.093,Z 370.819,A -85,B 0,C 180,E1 -19697.922,E2 -19697.922} C_VEL
LIN {X 0,Y 235.337,Z 370.789,A -85,B 0,C 180,E1 -19701.954,E2 -19701.954} C_VEL
LIN {X 0,Y 235.352,Z 370.864,A -85,B 0,C 180,E1 -19702.062,E2 -19702.062} C_VEL
LIN {X 0,Y 236.176,Z 373.38,A -85,B 0,C 180,E1 -19702.347,E2 -19702.347} C_VEL
LIN {X 0,Y 238.138,Z 376.003,A -85,B 0,C 180,E1 -19702.872,E2 -19702.872} C_VEL
LIN {X 0,Y 245.305,Z 387.368,A -85,B 0,C 180,E1 -19704.768,E2 -19704.768} C_VEL
LIN {X 0,Y 251.792,Z 397.951,A -85,B 0,C 180,E1 -19706.368,E2 -19706.368} C_VEL
LIN {X 0,Y 257.672,Z 408.967,A -85,B 0,C 180,E1 -19707.803,E2 -19707.803} C_VEL
LIN {X 0,Y 266.382,Z 425.569,A -85,B 0,C 180,E1 -19709.779,E2 -19709.779} C_VEL
LIN {X 0,Y 267.77,Z 428.511,A -85,B 0,C 180,E1 -19710.093,E2 -19710.093} C_VEL
LIN {X 0,Y 262.56,Z 522.283,A -85,B 0,C 180,E1 -19712.782,E2 -19712.782} C_VEL
LIN {X 0,Y 261.087,Z 538.128,A -85,B 0,C 180,E1 -19713.528,E2 -19713.528} C_VEL
LIN {X 0,Y 259.267,Z 553.009,A -85,B 0,C 180,E1 -19714.535,E2 -19714.535} C_VEL
LIN {X 0,Y 256.771,Z 568.222,A -85,B 0,C 180,E1 -19715.892,E2 -19715.892} C_VEL
LIN {X 0,Y 254.059,Z 582.301,A -85,B 0,C 180,E1 -19717.506,E2 -19717.506} C_VEL
LIN {X 0,Y 251.296,Z 594.684,A -85,B 0,C 180,E1 -19719.255,E2 -19719.255} C_VEL
LIN {X 0,Y 248.183,Z 607.239,A -85,B 0,C 180,E1 -19721.434,E2 -19721.434} C_VEL
LIN {X 0,Y 245.059,Z 618.887,A -85,B 0,C 180,E1 -19723.916,E2 -19723.916} C_VEL
LIN {X 0,Y 242.095,Z 629.408,A -85,B 0,C 180,E1 -19726.665,E2 -19726.665} C_VEL
LIN {X 0,Y 239.683,Z 637.899,A -85,B 0,C 180,E1 -19729.358,E2 -19729.358} C_VEL
LIN {X 0,Y 237.344,Z 646.282,A -85,B 0,C 180,E1 -19732.641,E2 -19732.641} C_VEL
LIN {X 0,Y 235.751,Z 652.196,A -85,B 0,C 180,E1 -19735.501,E2 -19735.501} C_VEL
LIN {X 0,Y 234.525,Z 657.392,A -85,B 0,C 180,E1 -19738.652,E2 -19738.652} C_VEL
LIN {X 0,Y 233.675,Z 661.222,A -85,B 0,C 180,E1 -19741.617,E2 -19741.617} C_VEL
LIN {X 0,Y 232.864,Z 664.735,A -85,B 0,C 180,E1 -19745.423,E2 -19745.423} C_VEL
LIN {X 0,Y 232.657,Z 666.402,A -85,B 0,C 180,E1 -19748.242,E2 -19748.242} C_VEL
LIN {X 0,Y 232.73,Z 667.36,A -85,B 0,C 180,E1 -19751.634,E2 -19751.634} C_VEL
LIN {X 0,Y 232.951,Z 667.413,A -85,B 0,C 180,E1 -19753.94,E2 -19753.94} C_VEL
LIN {X 0,Y 233.371,Z 666.959,A -85,B 0,C 180,E1 -19756.284,E2 -19756.284} C_VEL
LIN {X 0,Y 234.404,Z 665.193,A -85,B 0,C 180,E1 -19759.868,E2 -19759.868} C_VEL
LIN {X 0,Y 235.993,Z 662.069,A -85,B 0,C 180,E1 -19763.522,E2 -19763.522} C_VEL
LIN {X 0,Y 238.136,Z 657.732,A -85,B 0,C 180,E1 -19767.008,E2 -19767.008} C_VEL
LIN {X 0,Y 240.804,Z 652.331,A -85,B 0,C 180,E1 -19770.253,E2 -19770.253} C_VEL
LIN {X 0,Y 243.929,Z 645.9,A -85,B 0,C 180,E1 -19773.275,E2 -19773.275} C_VEL
LIN {X 0,Y 247.548,Z 638.24,A -85,B 0,C 180,E1 -19776.146,E2 -19776.146} C_VEL
LIN {X 0,Y 252.049,Z 628.245,A -85,B 0,C 180,E1 -19779.133,E2 -19779.133} C_VEL
LIN {X 0,Y 256.241,Z 617.989,A -85,B 0,C 180,E1 -19781.614,E2 -19781.614} C_VEL
LIN {X 0,Y 260.386,Z 607.137,A -85,B 0,C 180,E1 -19783.737,E2 -19783.737} C_VEL
LIN {X 0,Y 264.338,Z 595.715,A -85,B 0,C 180,E1 -19785.566,E2 -19785.566} C_VEL
LIN {X 0,Y 268.287,Z 582.817,A -85,B 0,C 180,E1 -19787.238,E2 -19787.238} C_VEL
LIN {X 0,Y 271.356,Z 570.842,A -85,B 0,C 180,E1 -19788.533,E2 -19788.533} C_VEL
LIN {X 0,Y 274.553,Z 556.188,A -85,B 0,C 180,E1 -19789.765,E2 -19789.765} C_VEL
LIN {X 0,Y 277.068,Z 541.19,A -85,B 0,C 180,E1 -19790.723,E2 -19790.723} C_VEL
LIN {X 0,Y 278.881,Z 526.422,A -85,B 0,C 180,E1 -19791.39,E2 -19791.39} C_VEL
LIN {X 0,Y 284.961,Z 448.115,A -85,B 0,C 180,E1 -19793.618,E2 -19793.618} C_VEL
LIN {X 0,Y 285.508,Z 439.25,A -85,B 0,C 180,E1 -19793.908,E2 -19793.908} C_VEL
LIN {X 0,Y 280.986,Z 430.426,A -85,B 0,C 180,E1 -19795.666,E2 -19795.666} C_VEL
LIN {X 0,Y 275.084,Z 420.22,A -85,B 0,C 180,E1 -19798.191,E2 -19798.191} C_VEL
LIN {X 0,Y 273.809,Z 418.287,A -85,B 0,C 180,E1 -19798.769,E2 -19798.769} C_VEL
LIN {X 0,Y 271.696,Z 415.527,A -85,B 0,C 180,E1 -19799.767,E2 -19799.767} C_VEL
LIN {X 0,Y 269.347,Z 413.79,A -85,B 0,C 180,E1 -19800.859,E2 -19800.859} C_VEL
LIN {X 0,Y 261.846,Z 410.28,A -85,B 0,C 180,E1 -19804.819,E2 -19804.819} C_VEL
LIN {X 0,Y 259.22,Z 406.578,A -85,B 0,C 180,E1 -19806.821,E2 -19806.821} C_VEL
LIN {X 0,Y 256.537,Z 403.38,A -85,B 0,C 180,E1 -19809.262,E2 -19809.262} C_VEL
LIN {X 0,Y 255.679,Z 401.643,A -85,B 0,C 180,E1 -19810.251,E2 -19810.251} C_VEL
LIN {X 0,Y 252.845,Z 399.322,A -85,B 0,C 180,E1 -19814.183,E2 -19814.183} C_VEL
LIN {X 0,Y 251.928,Z 396.813,A -85,B 0,C 180,E1 -19817.454,E2 -19817.454} C_VEL
LIN {X 0,Y 251.664,Z 397.531,A -85,B 0,C 180,E1 -19820.921,E2 -19820.921} C_VEL
LIN {X 0,Y 252.84,Z 399.457,A -85,B 0,C 180,E1 -19824.979,E2 -19824.979} C_VEL
LIN {X 0,Y 256.018,Z 405.204,A -85,B 0,C 180,E1 -19829.682,E2 -19829.682} C_VEL
LIN {X 0,Y 257.708,Z 407.72,A -85,B 0,C 180,E1 -19831.356,E2 -19831.356} C_VEL
LIN {X 0,Y 261.452,Z 414.061,A -85,B 0,C 180,E1 -19834.454,E2 -19834.454} C_VEL
LIN {X 0,Y 265.135,Z 420.609,A -85,B 0,C 180,E1 -19836.908,E2 -19836.908} C_VEL
LIN {X 0,Y 268.03,Z 426.115,A -85,B 0,C 180,E1 -19838.61,E2 -19838.61} C_VEL
LIN {X 0,Y 272.253,Z 434.528,A -85,B 0,C 180,E1 -19840.824,E2 -19840.824} C_VEL
LIN {X 0,Y 276.635,Z 444.487,A -85,B 0,C 180,E1 -19842.904,E2 -19842.904} C_VEL
LIN {X 0,Y 280.396,Z 454.426,A -85,B 0,C 180,E1 -19844.572,E2 -19844.572} C_VEL
LIN {X 0,Y 280.424,Z 457.389,A -85,B 0,C 180,E1 -19844.733,E2 -19844.733} C_VEL
LIN {X 0,Y 273.269,Z 545.014,A -85,B 0,C 180,E1 -19847.224,E2 -19847.224} C_VEL
LIN {X 0,Y 270.931,Z 561.196,A -85,B 0,C 180,E1 -19847.902,E2 -19847.902} C_VEL
LIN {X 0,Y 267.939,Z 576.108,A -85,B 0,C 180,E1 -19848.774,E2 -19848.774} C_VEL
LIN {X 0,Y 264.407,Z 590.218,A -85,B 0,C 180,E1 -19849.866,E2 -19849.866} C_VEL
LIN {X 0,Y 260.084,Z 604.702,A -85,B 0,C 180,E1 -19851.326,E2 -19851.326} C_VEL
LIN {X 0,Y 255.619,Z 617.932,A -85,B 0,C 180,E1 -19853.036,E2 -19853.036} C_VEL
LIN {X 0,Y 251.092,Z 630.056,A -85,B 0,C 180,E1 -19854.984,E2 -19854.984} C_VEL
LIN {X 0,Y 246.476,Z 641.291,A -85,B 0,C 180,E1 -19857.195,E2 -19857.195} C_VEL
LIN {X 0,Y 241.68,Z 652.307,A -85,B 0,C 180,E1 -19859.892,E2 -19859.892} C_VEL
LIN {X 0,Y 237.615,Z 661.451,A -85,B 0,C 180,E1 -19862.687,E2 -19862.687} C_VEL
LIN {X 0,Y 233.641,Z 670.305,A -85,B 0,C 180,E1 -19866.04,E2 -19866.04} C_VEL
LIN {X 0,Y 230.484,Z 677.445,A -85,B 0,C 180,E1 -19869.471,E2 -19869.471} C_VEL
LIN {X 0,Y 228.143,Z 683.389,A -85,B 0,C 180,E1 -19873.165,E2 -19873.165} C_VEL
LIN {X 0,Y 227.048,Z 686.542,A -85,B 0,C 180,E1 -19875.662,E2 -19875.662} C_VEL
LIN {X 0,Y 226.046,Z 690.03,A -85,B 0,C 180,E1 -19879.248,E2 -19879.248} C_VEL
LIN {X 0,Y 225.774,Z 692.275,A -85,B 0,C 180,E1 -19882.847,E2 -19882.847} C_VEL
LIN {X 0,Y 225.845,Z 693.348,A -85,B 0,C 180,E1 -19886.431,E2 -19886.431} C_VEL
LIN {X 0,Y 225.997,Z 693.239,A -85,B 0,C 180,E1 -19889.999,E2 -19889.999} C_VEL
LIN {X 0,Y 225.886,Z 691.891,A -85,B 0,C 180,E1 -19893.567,E2 -19893.567} C_VEL
LIN {X 0,Y 225.88,Z 690.747,A -85,B 0,C 180,E1 -19895.355,E2 -19895.355} C_VEL
LIN {X 0,Y 225.919,Z 687.454,A -85,B 0,C 180,E1 -19898.947,E2 -19898.947} C_VEL
LIN {X 0,Y 226.421,Z 682.77,A -85,B 0,C 180,E1 -19902.548,E2 -19902.548} C_VEL
LIN {X 0,Y 227.622,Z 676.615,A -85,B 0,C 180,E1 -19906.133,E2 -19906.133} C_VEL
LIN {X 0,Y 229.514,Z 668.822,A -85,B 0,C 180,E1 -19909.683,E2 -19909.683} C_VEL
LIN {X 0,Y 231.86,Z 660.44,A -85,B 0,C 180,E1 -19912.734,E2 -19912.734} C_VEL
LIN {X 0,Y 234.471,Z 650.904,A -85,B 0,C 180,E1 -19915.58,E2 -19915.58} C_VEL
LIN {X 0,Y 237.6,Z 639.953,A -85,B 0,C 180,E1 -19918.246,E2 -19918.246} C_VEL
LIN {X 0,Y 240.989,Z 627.612,A -85,B 0,C 180,E1 -19920.687,E2 -19920.687} C_VEL
LIN {X 0,Y 244.317,Z 615.289,A -85,B 0,C 180,E1 -19922.639,E2 -19922.639} C_VEL
LIN {X 0,Y 247.455,Z 601.89,A -85,B 0,C 180,E1 -19924.365,E2 -19924.365} C_VEL
LIN {X 0,Y 250.376,Z 587.169,A -85,B 0,C 180,E1 -19925.869,E2 -19925.869} C_VEL
LIN {X 0,Y 253.049,Z 571.883,A -85,B 0,C 180,E1 -19927.036,E2 -19927.036} C_VEL
LIN {X 0,Y 254.976,Z 556.666,A -85,B 0,C 180,E1 -19927.889,E2 -19927.889} C_VEL
LIN {X 0,Y 256.225,Z 540.979,A -85,B 0,C 180,E1 -19928.483,E2 -19928.483} C_VEL
LIN {X 0,Y 261.282,Z 452.519,A -85,B 0,C 180,E1 -19931.04,E2 -19931.04} C_VEL
LIN {X 0,Y 259.756,Z 440.878,A -85,B 0,C 180,E1 -19931.705,E2 -19931.705} C_VEL
LIN {X 0,Y 252.318,Z 423.064,A -85,B 0,C 180,E1 -19933.599,E2 -19933.599} C_VEL
LIN {X 0,Y 243.406,Z 404.259,A -85,B 0,C 180,E1 -19935.953,E2 -19935.953} C_VEL
LIN {X 0,Y 235.563,Z 389.286,A -85,B 0,C 180,E1 -19938.144,E2 -19938.144} C_VEL
LIN {X 0,Y 231.722,Z 382.547,A -85,B 0,C 180,E1 -19939.259,E2 -19939.259} C_VEL
LIN {X 0,Y 230.362,Z 379.837,A -85,B 0,C 180,E1 -19939.703,E2 -19939.703} C_VEL
LIN {X 0,Y 227.884,Z 371.72,A -85,B 0,C 180,E1 -19943.189,E2 -19943.189} C_VEL
LIN {X 0,Y 227.876,Z 371.712,A -85,B 0,C 180,E1 -19946.377,E2 -19946.377} C_VEL
LIN {X 0,Y 227.916,Z 371.721,A -85,B 0,C 180,E1 -19950.438,E2 -19950.438} C_VEL
LIN {X 0,Y 227.926,Z 371.714,A -85,B 0,C 180,E1 -19954.426,E2 -19954.426} C_VEL
LIN {X 0,Y 227.959,Z 371.71,A -85,B 0,C 180,E1 -19958.287,E2 -19958.287} C_VEL
LIN {X 0,Y 228.032,Z 371.703,A -85,B 0,C 180,E1 -19962.826,E2 -19962.826} C_VEL
LIN {X 0,Y 228.072,Z 371.675,A -85,B 0,C 180,E1 -19967.544,E2 -19967.544} C_VEL
LIN {X 0,Y 228.302,Z 371.65,A -85,B 0,C 180,E1 -19971.147,E2 -19971.147} C_VEL
LIN {X 0,Y 228.351,Z 371.66,A -85,B 0,C 180,E1 -19972.929,E2 -19972.929} C_VEL
LIN {X 0,Y 228.553,Z 371.62,A -85,B 0,C 180,E1 -19978.239,E2 -19978.239} C_VEL
LIN {X 0,Y 228.553,Z 371.638,A -85,B 0,C 180,E1 -19981.763,E2 -19981.763} C_VEL
LIN {X 0,Y 228.356,Z 371.642,A -85,B 0,C 180,E1 -19987.072,E2 -19987.072} C_VEL
LIN {X 0,Y 228.17,Z 371.686,A -85,B 0,C 180,E1 -19990.651,E2 -19990.651} C_VEL
LIN {X 0,Y 228.056,Z 371.678,A -85,B 0,C 180,E1 -19996.103,E2 -19996.103} C_VEL
LIN {X 0,Y 227.936,Z 371.714,A -85,B 0,C 180,E1 -19999.827,E2 -19999.827} C_VEL
LIN {X 0,Y 227.905,Z 371.712,A -85,B 0,C 180,E1 -20003.634,E2 -20003.634} C_VEL
LIN {X 0,Y 227.885,Z 371.711,A -85,B 0,C 180,E1 -20007.556,E2 -20007.556} C_VEL
LIN {X 0,Y 227.87,Z 371.723,A -85,B 0,C 180,E1 -20011.623,E2 -20011.623} C_VEL
LIN {X 0,Y 227.879,Z 371.705,A -85,B 0,C 180,E1 -20015.873,E2 -20015.873} C_VEL
LIN {X 0,Y 227.824,Z 371.73,A -85,B 0,C 180,E1 -20020.378,E2 -20020.378} C_VEL
LIN {X 0,Y 227.826,Z 371.72,A -85,B 0,C 180,E1 -20025.196,E2 -20025.196} C_VEL
LIN {X 0,Y 227.825,Z 371.725,A -85,B 0,C 180,E1 -20029.624,E2 -20029.624} C_VEL
LIN {X 0,Y 227.882,Z 371.723,A -85,B 0,C 180,E1 -20034.13,E2 -20034.13} C_VEL
LIN {X 0,Y 227.857,Z 371.713,A -85,B 0,C 180,E1 -20038.377,E2 -20038.377} C_VEL
LIN {X 0,Y 227.858,Z 371.724,A -85,B 0,C 180,E1 -20042.442,E2 -20042.442} C_VEL
LIN {X 0,Y 227.897,Z 371.721,A -85,B 0,C 180,E1 -20046.366,E2 -20046.366} C_VEL
LIN {X 0,Y 227.915,Z 371.71,A -85,B 0,C 180,E1 -20050.173,E2 -20050.173} C_VEL
LIN {X 0,Y 228.003,Z 371.701,A -85,B 0,C 180,E1 -20053.895,E2 -20053.895} C_VEL
LIN {X 0,Y 228.143,Z 371.689,A -85,B 0,C 180,E1 -20059.35,E2 -20059.35} C_VEL
LIN {X 0,Y 228.25,Z 371.685,A -85,B 0,C 180,E1 -20060.566,E2 -20060.566} C_VEL
LIN {X 0,Y 229.241,Z 374.481,A -85,B 0,C 180,E1 -20060.922,E2 -20060.922} C_VEL
LIN {X 0,Y 231.156,Z 376.973,A -85,B 0,C 180,E1 -20061.459,E2 -20061.459} C_VEL
LIN {X 0,Y 233.41,Z 380.384,A -85,B 0,C 180,E1 -20062.096,E2 -20062.096} C_VEL
LIN {X 0,Y 245.414,Z 399.569,A -85,B 0,C 180,E1 -20065.305,E2 -20065.305} C_VEL
LIN {X 0,Y 251.957,Z 411.569,A -85,B 0,C 180,E1 -20066.946,E2 -20066.946} C_VEL
LIN {X 0,Y 261.291,Z 429.582,A -85,B 0,C 180,E1 -20069.163,E2 -20069.163} C_VEL
LIN {X 0,Y 261.793,Z 430.749,A -85,B 0,C 180,E1 -20069.284,E2 -20069.284} C_VEL
LIN {X 0,Y 256.507,Z 522.403,A -85,B 0,C 180,E1 -20071.963,E2 -20071.963} C_VEL
LIN {X 0,Y 255.004,Z 538.206,A -85,B 0,C 180,E1 -20072.716,E2 -20072.716} C_VEL
LIN {X 0,Y 253.098,Z 553.359,A -85,B 0,C 180,E1 -20073.76,E2 -20073.76} C_VEL
LIN {X 0,Y 250.717,Z 567.505,A -85,B 0,C 180,E1 -20075.026,E2 -20075.026} C_VEL
LIN {X 0,Y 247.985,Z 581.53,A -85,B 0,C 180,E1 -20076.638,E2 -20076.638} C_VEL
LIN {X 0,Y 245.051,Z 594.31,A -85,B 0,C 180,E1 -20078.453,E2 -20078.453} C_VEL
LIN {X 0,Y 241.899,Z 606.665,A -85,B 0,C 180,E1 -20080.611,E2 -20080.611} C_VEL
LIN {X 0,Y 238.808,Z 618.051,A -85,B 0,C 180,E1 -20083.049,E2 -20083.049} C_VEL
LIN {X 0,Y 235.992,Z 627.681,A -85,B 0,C 180,E1 -20085.548,E2 -20085.548} C_VEL
LIN {X 0,Y 233.231,Z 636.908,A -85,B 0,C 180,E1 -20088.446,E2 -20088.446} C_VEL
LIN {X 0,Y 230.695,Z 645.784,A -85,B 0,C 180,E1 -20091.902,E2 -20091.902} C_VEL
LIN {X 0,Y 228.626,Z 653.054,A -85,B 0,C 180,E1 -20095.491,E2 -20095.491} C_VEL
LIN {X 0,Y 227.441,Z 657.977,A -85,B 0,C 180,E1 -20098.618,E2 -20098.618} C_VEL
LIN {X 0,Y 226.495,Z 661.932,A -85,B 0,C 180,E1 -20101.837,E2 -20101.837} C_VEL
LIN {X 0,Y 225.992,Z 664.032,A -85,B 0,C 180,E1 -20104.041,E2 -20104.041} C_VEL
LIN {X 0,Y 225.669,Z 665.693,A -85,B 0,C 180,E1 -20106.28,E2 -20106.28} C_VEL
LIN {X 0,Y 225.547,Z 667.029,A -85,B 0,C 180,E1 -20108.83,E2 -20108.83} C_VEL
LIN {X 0,Y 225.652,Z 667.749,A -85,B 0,C 180,E1 -20111.626,E2 -20111.626} C_VEL
LIN {X 0,Y 226.14,Z 667.622,A -85,B 0,C 180,E1 -20115.628,E2 -20115.628} C_VEL
LIN {X 0,Y 227.175,Z 666.139,A -85,B 0,C 180,E1 -20119.483,E2 -20119.483} C_VEL
LIN {X 0,Y 228.648,Z 663.55,A -85,B 0,C 180,E1 -20123.052,E2 -20123.052} C_VEL
LIN {X 0,Y 230.844,Z 659.48,A -85,B 0,C 180,E1 -20126.769,E2 -20126.769} C_VEL
LIN {X 0,Y 233.341,Z 654.805,A -85,B 0,C 180,E1 -20129.928,E2 -20129.928} C_VEL
LIN {X 0,Y 237.087,Z 647.618,A -85,B 0,C 180,E1 -20133.598,E2 -20133.598} C_VEL
LIN {X 0,Y 241.198,Z 639.438,A -85,B 0,C 180,E1 -20136.835,E2 -20136.835} C_VEL
LIN {X 0,Y 245.215,Z 631.185,A -85,B 0,C 180,E1 -20139.445,E2 -20139.445} C_VEL
LIN {X 0,Y 249.417,Z 621.572,A -85,B 0,C 180,E1 -20141.943,E2 -20141.943} C_VEL
LIN {X 0,Y 253.721,Z 611.073,A -85,B 0,C 180,E1 -20144.151,E2 -20144.151} C_VEL
LIN {X 0,Y 257.994,Z 599.728,A -85,B 0,C 180,E1 -20146.105,E2 -20146.105} C_VEL
LIN {X 0,Y 261.909,Z 587.852,A -85,B 0,C 180,E1 -20147.789,E2 -20147.789} C_VEL
LIN {X 0,Y 265.749,Z 574.372,A -85,B 0,C 180,E1 -20149.331,E2 -20149.331} C_VEL
LIN {X 0,Y 269.119,Z 560.168,A -85,B 0,C 180,E1 -20150.606,E2 -20150.606} C_VEL
LIN {X 0,Y 271.853,Z 545.319,A -85,B 0,C 180,E1 -20151.638,E2 -20151.638} C_VEL
LIN {X 0,Y 274.006,Z 529.601,A -85,B 0,C 180,E1 -20152.423,E2 -20152.423} C_VEL
LIN {X 0,Y 275.963,Z 507.038,A -85,B 0,C 180,E1 -20153.143,E2 -20153.143} C_VEL
LIN {X 0,Y 281.228,Z 442.514,A -85,B 0,C 180,E1 -20154.958,E2 -20154.958} C_VEL
LIN {X 0,Y 276.433,Z 433.266,A -85,B 0,C 180,E1 -20156.962,E2 -20156.962} C_VEL
LIN {X 0,Y 271.958,Z 425.442,A -85,B 0,C 180,E1 -20159.014,E2 -20159.014} C_VEL
LIN {X 0,Y 265.557,Z 415.206,A -85,B 0,C 180,E1 -20162.466,E2 -20162.466} C_VEL
LIN {X 0,Y 262.696,Z 411.122,A -85,B 0,C 180,E1 -20164.272,E2 -20164.272} C_VEL
LIN {X 0,Y 261.846,Z 410.28,A -85,B 0,C 180,E1 -20164.819,E2 -20164.819} C_VEL
LIN {X 0,Y 259.423,Z 408.926,A -85,B 0,C 180,E1 -20166.44,E2 -20166.44} C_VEL
LIN {X 0,Y 253.453,Z 408.01,A -85,B 0,C 180,E1 -20171.582,E2 -20171.582} C_VEL
LIN {X 0,Y 251.25,Z 405.428,A -85,B 0,C 180,E1 -20175.483,E2 -20175.483} C_VEL
LIN {X 0,Y 250.808,Z 403.845,A -85,B 0,C 180,E1 -20177.685,E2 -20177.685} C_VEL
LIN {X 0,Y 250.608,Z 404.614,A -85,B 0,C 180,E1 -20181.014,E2 -20181.014} C_VEL
LIN {X 0,Y 251.605,Z 406.287,A -85,B 0,C 180,E1 -20184.634,E2 -20184.634} C_VEL
LIN {X 0,Y 254.832,Z 412.366,A -85,B 0,C 180,E1 -20189.614,E2 -20189.614} C_VEL
LIN {X 0,Y 256.052,Z 414.314,A -85,B 0,C 180,E1 -20190.876,E2 -20190.876} C_VEL
LIN {X 0,Y 259.429,Z 420.267,A -85,B 0,C 180,E1 -20193.839,E2 -20193.839} C_VEL
LIN {X 0,Y 262.911,Z 426.77,A -85,B 0,C 180,E1 -20196.308,E2 -20196.308} C_VEL
LIN {X 0,Y 266.313,Z 433.538,A -85,B 0,C 180,E1 -20198.403,E2 -20198.403} C_VEL
LIN {X 0,Y 270.58,Z 442.761,A -85,B 0,C 180,E1 -20200.723,E2 -20200.723} C_VEL
LIN {X 0,Y 273.913,Z 451.012,A -85,B 0,C 180,E1 -20202.377,E2 -20202.377} C_VEL
LIN {X 0,Y 276.276,Z 457.421,A -85,B 0,C 180,E1 -20203.505,E2 -20203.505} C_VEL
LIN {X 0,Y 271.378,Z 516.672,A -85,B 0,C 180,E1 -20205.2,E2 -20205.2} C_VEL
LIN {X 0,Y 268.796,Z 545.833,A -85,B 0,C 180,E1 -20206.076,E2 -20206.076} C_VEL
LIN {X 0,Y 266.366,Z 561.522,A -85,B 0,C 180,E1 -20206.75,E2 -20206.75} C_VEL
LIN {X 0,Y 263.261,Z 576.163,A -85,B 0,C 180,E1 -20207.617,E2 -20207.617} C_VEL
LIN {X 0,Y 259.611,Z 590.1,A -85,B 0,C 180,E1 -20208.71,E2 -20208.71} C_VEL
LIN {X 0,Y 255.126,Z 604.526,A -85,B 0,C 180,E1 -20210.172,E2 -20210.172} C_VEL
LIN {X 0,Y 250.532,Z 617.664,A -85,B 0,C 180,E1 -20211.891,E2 -20211.891} C_VEL
LIN {X 0,Y 245.766,Z 629.78,A -85,B 0,C 180,E1 -20213.856,E2 -20213.856} C_VEL
LIN {X 0,Y 240.565,Z 641.772,A -85,B 0,C 180,E1 -20216.283,E2 -20216.283} C_VEL
LIN {X 0,Y 236.233,Z 651.173,A -85,B 0,C 180,E1 -20218.625,E2 -20218.625} C_VEL
LIN {X 0,Y 232.415,Z 659.244,A -85,B 0,C 180,E1 -20221.064,E2 -20221.064} C_VEL
LIN {X 0,Y 228.633,Z 667.295,A -85,B 0,C 180,E1 -20224.021,E2 -20224.021} C_VEL
LIN {X 0,Y 225.325,Z 674.063,A -85,B 0,C 180,E1 -20227.052,E2 -20227.052} C_VEL
LIN {X 0,Y 222.487,Z 680.374,A -85,B 0,C 180,E1 -20230.629,E2 -20230.629} C_VEL
LIN {X 0,Y 220.452,Z 685.31,A -85,B 0,C 180,E1 -20234.277,E2 -20234.277} C_VEL
LIN {X 0,Y 219.428,Z 688.187,A -85,B 0,C 180,E1 -20237.043,E2 -20237.043} C_VEL
LIN {X 0,Y 218.765,Z 690.999,A -85,B 0,C 180,E1 -20240.756,E2 -20240.756} C_VEL
LIN {X 0,Y 218.712,Z 692.743,A -85,B 0,C 180,E1 -20244.96,E2 -20244.96} C_VEL
LIN {X 0,Y 218.848,Z 693.01,A -85,B 0,C 180,E1 -20248.159,E2 -20248.159} C_VEL
LIN {X 0,Y 218.922,Z 692.769,A -85,B 0,C 180,E1 -20249.999,E2 -20249.999} C_VEL
LIN {X 0,Y 218.805,Z 691.348,A -85,B 0,C 180,E1 -20253.682,E2 -20253.682} C_VEL
LIN {X 0,Y 218.796,Z 690.166,A -85,B 0,C 180,E1 -20255.529,E2 -20255.529} C_VEL
LIN {X 0,Y 218.868,Z 686.808,A -85,B 0,C 180,E1 -20259.238,E2 -20259.238} C_VEL
LIN {X 0,Y 219.431,Z 682.058,A -85,B 0,C 180,E1 -20262.955,E2 -20262.955} C_VEL
LIN {X 0,Y 220.722,Z 675.812,A -85,B 0,C 180,E1 -20266.652,E2 -20266.652} C_VEL
LIN {X 0,Y 222.436,Z 668.964,A -85,B 0,C 180,E1 -20269.855,E2 -20269.855} C_VEL
LIN {X 0,Y 224.845,Z 660.701,A -85,B 0,C 180,E1 -20272.998,E2 -20272.998} C_VEL
LIN {X 0,Y 227.29,Z 652.255,A -85,B 0,C 180,E1 -20275.65,E2 -20275.65} C_VEL
LIN {X 0,Y 230.184,Z 642.326,A -85,B 0,C 180,E1 -20278.244,E2 -20278.244} C_VEL
LIN {X 0,Y 233.64,Z 630.536,A -85,B 0,C 180,E1 -20280.754,E2 -20280.754} C_VEL
LIN {X 0,Y 236.829,Z 618.842,A -85,B 0,C 180,E1 -20282.79,E2 -20282.79} C_VEL
LIN {X 0,Y 240.089,Z 606.335,A -85,B 0,C 180,E1 -20284.551,E2 -20284.551} C_VEL
LIN {X 0,Y 243.159,Z 591.88,A -85,B 0,C 180,E1 -20286.192,E2 -20286.192} C_VEL
LIN {X 0,Y 245.834,Z 577.927,A -85,B 0,C 180,E1 -20287.408,E2 -20287.408} C_VEL
LIN {X 0,Y 248.161,Z 562.545,A -85,B 0,C 180,E1 -20288.408,E2 -20288.408} C_VEL
LIN {X 0,Y 249.77,Z 547.788,A -85,B 0,C 180,E1 -20289.083,E2 -20289.083} C_VEL
LIN {X 0,Y 255.351,Z 452.975,A -85,B 0,C 180,E1 -20291.922,E2 -20291.922} C_VEL
LIN {X 0,Y 253.93,Z 443.041,A -85,B 0,C 180,E1 -20292.537,E2 -20292.537} C_VEL
LIN {X 0,Y 246.01,Z 424.221,A -85,B 0,C 180,E1 -20294.642,E2 -20294.642} C_VEL
LIN {X 0,Y 237.974,Z 407.24,A -85,B 0,C 180,E1 -20296.854,E2 -20296.854} C_VEL
LIN {X 0,Y 230.624,Z 393.18,A -85,B 0,C 180,E1 -20298.995,E2 -20298.995} C_VEL
LIN {X 0,Y 225.052,Z 383.241,A -85,B 0,C 180,E1 -20300.703,E2 -20300.703} C_VEL
LIN {X 0,Y 222.918,Z 379.315,A -85,B 0,C 180,E1 -20301.425,E2 -20301.425} C_VEL
LIN {X 0,Y 220.831,Z 372.608,A -85,B 0,C 180,E1 -20304.493,E2 -20304.493} C_VEL
LIN {X 0,Y 220.865,Z 372.604,A -85,B 0,C 180,E1 -20309.395,E2 -20309.395} C_VEL
LIN {X 0,Y 220.892,Z 372.591,A -85,B 0,C 180,E1 -20313.55,E2 -20313.55} C_VEL
LIN {X 0,Y 220.875,Z 372.591,A -85,B 0,C 180,E1 -20317.554,E2 -20317.554} C_VEL
LIN {X 0,Y 220.981,Z 372.579,A -85,B 0,C 180,E1 -20322.571,E2 -20322.571} C_VEL
LIN {X 0,Y 221.011,Z 372.558,A -85,B 0,C 180,E1 -20327.139,E2 -20327.139} C_VEL
LIN {X 0,Y 221.233,Z 372.526,A -85,B 0,C 180,E1 -20330.861,E2 -20330.861} C_VEL
LIN {X 0,Y 221.286,Z 372.538,A -85,B 0,C 180,E1 -20332.702,E2 -20332.702} C_VEL
LIN {X 0,Y 221.511,Z 372.496,A -85,B 0,C 180,E1 -20338.182,E2 -20338.182} C_VEL
LIN {X 0,Y 221.511,Z 372.516,A -85,B 0,C 180,E1 -20341.819,E2 -20341.819} C_VEL
LIN {X 0,Y 221.293,Z 372.521,A -85,B 0,C 180,E1 -20347.299,E2 -20347.299} C_VEL
LIN {X 0,Y 221.115,Z 372.567,A -85,B 0,C 180,E1 -20350.995,E2 -20350.995} C_VEL
LIN {X 0,Y 221.015,Z 372.554,A -85,B 0,C 180,E1 -20356.631,E2 -20356.631} C_VEL
LIN {X 0,Y 220.883,Z 372.594,A -85,B 0,C 180,E1 -20360.488,E2 -20360.488} C_VEL
LIN {X 0,Y 220.861,Z 372.578,A -85,B 0,C 180,E1 -20364.437,E2 -20364.437} C_VEL
LIN {X 0,Y 220.836,Z 372.594,A -85,B 0,C 180,E1 -20368.515,E2 -20368.515} C_VEL
LIN {X 0,Y 220.817,Z 372.593,A -85,B 0,C 180,E1 -20372.757,E2 -20372.757} C_VEL
LIN {X 0,Y 220.81,Z 372.597,A -85,B 0,C 180,E1 -20377.279,E2 -20377.279} C_VEL
LIN {X 0,Y 220.794,Z 372.607,A -85,B 0,C 180,E1 -20380.189,E2 -20380.189} C_VEL
LIN {X 0,Y 220.767,Z 372.591,A -85,B 0,C 180,E1 -20384.457,E2 -20384.457} C_VEL
LIN {X 0,Y 220.767,Z 372.611,A -85,B 0,C 180,E1 -20388.048,E2 -20388.048} C_VEL
LIN {X 0,Y 220.807,Z 372.59,A -85,B 0,C 180,E1 -20390.464,E2 -20390.464} C_VEL
LIN {X 0,Y 220.802,Z 372.607,A -85,B 0,C 180,E1 -20395.046,E2 -20395.046} C_VEL
LIN {X 0,Y 220.835,Z 372.592,A -85,B 0,C 180,E1 -20399.391,E2 -20399.391} C_VEL
LIN {X 0,Y 220.878,Z 372.586,A -85,B 0,C 180,E1 -20403.548,E2 -20403.548} C_VEL
LIN {X 0,Y 220.87,Z 372.597,A -85,B 0,C 180,E1 -20407.553,E2 -20407.553} C_VEL
LIN {X 0,Y 220.921,Z 372.59,A -85,B 0,C 180,E1 -20412.627,E2 -20412.627} C_VEL
LIN {X 0,Y 220.981,Z 372.581,A -85,B 0,C 180,E1 -20417.138,E2 -20417.138} C_VEL
LIN {X 0,Y 221.076,Z 372.565,A -85,B 0,C 180,E1 -20418.889,E2 -20418.889} C_VEL
LIN {X 0,Y 222.145,Z 375.488,A -85,B 0,C 180,E1 -20419.332,E2 -20419.332} C_VEL
LIN {X 0,Y 224.166,Z 377.834,A -85,B 0,C 180,E1 -20419.93,E2 -20419.93} C_VEL
LIN {X 0,Y 226.546,Z 381.418,A -85,B 0,C 180,E1 -20420.654,E2 -20420.654} C_VEL
LIN {X 0,Y 240.677,Z 403.931,A -85,B 0,C 180,E1 -20424.607,E2 -20424.607} C_VEL
LIN {X 0,Y 246.951,Z 415.559,A -85,B 0,C 180,E1 -20426.246,E2 -20426.246} C_VEL
LIN {X 0,Y 255.809,Z 432.801,A -85,B 0,C 180,E1 -20428.426,E2 -20428.426} C_VEL
LIN {X 0,Y 250.514,Z 522.427,A -85,B 0,C 180,E1 -20431.106,E2 -20431.106} C_VEL
LIN {X 0,Y 248.963,Z 538.354,A -85,B 0,C 180,E1 -20431.871,E2 -20431.871} C_VEL
LIN {X 0,Y 246.897,Z 554.096,A -85,B 0,C 180,E1 -20432.978,E2 -20432.978} C_VEL
LIN {X 0,Y 244.353,Z 568.709,A -85,B 0,C 180,E1 -20434.331,E2 -20434.331} C_VEL
LIN {X 0,Y 241.731,Z 581.608,A -85,B 0,C 180,E1 -20435.841,E2 -20435.841} C_VEL
LIN {X 0,Y 238.494,Z 595.279,A -85,B 0,C 180,E1 -20437.834,E2 -20437.834} C_VEL
LIN {X 0,Y 235.235,Z 607.559,A -85,B 0,C 180,E1 -20440.046,E2 -20440.046} C_VEL
LIN {X 0,Y 232.014,Z 619.012,A -85,B 0,C 180,E1 -20442.584,E2 -20442.584} C_VEL
LIN {X 0,Y 228.63,Z 630.086,A -85,B 0,C 180,E1 -20445.604,E2 -20445.604} C_VEL
LIN {X 0,Y 225.908,Z 638.994,A -85,B 0,C 180,E1 -20448.596,E2 -20448.596} C_VEL
LIN {X 0,Y 223.67,Z 646.48,A -85,B 0,C 180,E1 -20451.667,E2 -20451.667} C_VEL
LIN {X 0,Y 221.566,Z 653.661,A -85,B 0,C 180,E1 -20455.355,E2 -20455.355} C_VEL
LIN {X 0,Y 220.337,Z 658.565,A -85,B 0,C 180,E1 -20458.585,E2 -20458.585} C_VEL
LIN {X 0,Y 219.369,Z 662.482,A -85,B 0,C 180,E1 -20461.913,E2 -20461.913} C_VEL
LIN {X 0,Y 218.676,Z 665.445,A -85,B 0,C 180,E1 -20465.346,E2 -20465.346} C_VEL
LIN {X 0,Y 218.469,Z 667.592,A -85,B 0,C 180,E1 -20469.459,E2 -20469.459} C_VEL
LIN {X 0,Y 218.632,Z 668.253,A -85,B 0,C 180,E1 -20472.459,E2 -20472.459} C_VEL
LIN {X 0,Y 218.967,Z 668.245,A -85,B 0,C 180,E1 -20475.079,E2 -20475.079} C_VEL
LIN {X 0,Y 219.56,Z 667.58,A -85,B 0,C 180,E1 -20477.762,E2 -20477.762} C_VEL
LIN {X 0,Y 220.392,Z 666.376,A -85,B 0,C 180,E1 -20480.373,E2 -20480.373} C_VEL
LIN {X 0,Y 222.097,Z 663.596,A -85,B 0,C 180,E1 -20484.115,E2 -20484.115} C_VEL
LIN {X 0,Y 224.498,Z 659.475,A -85,B 0,C 180,E1 -20487.846,E2 -20487.846} C_VEL
LIN {X 0,Y 227.591,Z 654.053,A -85,B 0,C 180,E1 -20491.444,E2 -20491.444} C_VEL
LIN {X 0,Y 231.295,Z 647.391,A -85,B 0,C 180,E1 -20494.824,E2 -20494.824} C_VEL
LIN {X 0,Y 235.287,Z 639.908,A -85,B 0,C 180,E1 -20497.817,E2 -20497.817} C_VEL
LIN {X 0,Y 239.906,Z 630.73,A -85,B 0,C 180,E1 -20500.739,E2 -20500.739} C_VEL
LIN {X 0,Y 244.434,Z 620.915,A -85,B 0,C 180,E1 -20503.29,E2 -20503.29} C_VEL
LIN {X 0,Y 248.938,Z 610.425,A -85,B 0,C 180,E1 -20505.489,E2 -20505.489} C_VEL
LIN {X 0,Y 253.823,Z 597.825,A -85,B 0,C 180,E1 -20507.608,E2 -20507.608} C_VEL
LIN {X 0,Y 258.217,Z 584.687,A -85,B 0,C 180,E1 -20509.382,E2 -20509.382} C_VEL
LIN {X 0,Y 261.646,Z 572.545,A -85,B 0,C 180,E1 -20510.725,E2 -20510.725} C_VEL
LIN {X 0,Y 265.184,Z 557.855,A -85,B 0,C 180,E1 -20511.994,E2 -20511.994} C_VEL
LIN {X 0,Y 267.863,Z 543.391,A -85,B 0,C 180,E1 -20512.953,E2 -20512.953} C_VEL
LIN {X 0,Y 269.864,Z 528.675,A -85,B 0,C 180,E1 -20513.657,E2 -20513.657} C_VEL
LIN {X 0,Y 272.861,Z 493.743,A -85,B 0,C 180,E1 -20514.719,E2 -20514.719} C_VEL
LIN {X 0,Y 276.93,Z 445.646,A -85,B 0,C 180,E1 -20516.091,E2 -20516.091} C_VEL
LIN {X 0,Y 271.413,Z 434.981,A -85,B 0,C 180,E1 -20518.609,E2 -20518.609} C_VEL
LIN {X 0,Y 268.11,Z 429.355,A -85,B 0,C 180,E1 -20520.289,E2 -20520.289} C_VEL
LIN {X 0,Y 263.095,Z 421.093,A -85,B 0,C 180,E1 -20523.213,E2 -20523.213} C_VEL
LIN {X 0,Y 260.661,Z 417.515,A -85,B 0,C 180,E1 -20524.839,E2 -20524.839} C_VEL
LIN {X 0,Y 257.474,Z 413.16,A -85,B 0,C 180,E1 -20527.33,E2 -20527.33} C_VEL
LIN {X 0,Y 254.927,Z 409.878,A -85,B 0,C 180,E1 -20529.784,E2 -20529.784} C_VEL
LIN {X 0,Y 254.243,Z 408.503,A -85,B 0,C 180,E1 -20530.638,E2 -20530.638} C_VEL
LIN {X 0,Y 253.453,Z 408.01,A -85,B 0,C 180,E1 -20531.582,E2 -20531.582} C_VEL
LIN {X 0,Y 252.09,Z 408.014,A -85,B 0,C 180,E1 -20533.342,E2 -20533.342} C_VEL
LIN {X 0,Y 249.753,Z 410.721,A -85,B 0,C 180,E1 -20537.798,E2 -20537.798} C_VEL
LIN {X 0,Y 249.565,Z 410.998,A -85,B 0,C 180,E1 -20538.705,E2 -20538.705} C_VEL
LIN {X 0,Y 250.124,Z 412.721,A -85,B 0,C 180,E1 -20543.602,E2 -20543.602} C_VEL
LIN {X 0,Y 250.643,Z 413.941,A -85,B 0,C 180,E1 -20544.989,E2 -20544.989} C_VEL
LIN {X 0,Y 253.96,Z 419.943,A -85,B 0,C 180,E1 -20549.875,E2 -20549.875} C_VEL
LIN {X 0,Y 257.488,Z 426.572,A -85,B 0,C 180,E1 -20553.251,E2 -20553.251} C_VEL
LIN {X 0,Y 260.489,Z 432.493,A -85,B 0,C 180,E1 -20555.542,E2 -20555.542} C_VEL
LIN {X 0,Y 263.187,Z 438.091,A -85,B 0,C 180,E1 -20557.337,E2 -20557.337} C_VEL
LIN {X 0,Y 266.955,Z 446.521,A -85,B 0,C 180,E1 -20559.56,E2 -20559.56} C_VEL
LIN {X 0,Y 270.231,Z 454.758,A -85,B 0,C 180,E1 -20561.331,E2 -20561.331} C_VEL
LIN {X 0,Y 272.221,Z 460.377,A -85,B 0,C 180,E1 -20562.356,E2 -20562.356} C_VEL
LIN {X 0,Y 264.669,Z 544.813,A -85,B 0,C 180,E1 -20564.806,E2 -20564.806} C_VEL
LIN {X 0,Y 262.188,Z 560.637,A -85,B 0,C 180,E1 -20565.482,E2 -20565.482} C_VEL
LIN {X 0,Y 258.975,Z 575.378,A -85,B 0,C 180,E1 -20566.344,E2 -20566.344} C_VEL
LIN {X 0,Y 254.945,Z 590.22,A -85,B 0,C 180,E1 -20567.515,E2 -20567.515} C_VEL
LIN {X 0,Y 250.293,Z 604.464,A -85,B 0,C 180,E1 -20568.977,E2 -20568.977} C_VEL
LIN {X 0,Y 245.49,Z 617.479,A -85,B 0,C 180,E1 -20570.7,E2 -20570.7} C_VEL
LIN {X 0,Y 240.539,Z 629.529,A -85,B 0,C 180,E1 -20572.679,E2 -20572.679} C_VEL
LIN {X 0,Y 235.53,Z 640.668,A -85,B 0,C 180,E1 -20574.941,E2 -20574.941} C_VEL
LIN {X 0,Y 230.185,Z 651.588,A -85,B 0,C 180,E1 -20577.702,E2 -20577.702} C_VEL
LIN {X 0,Y 225.259,Z 661.454,A -85,B 0,C 180,E1 -20580.878,E2 -20580.878} C_VEL
LIN {X 0,Y 221.702,Z 668.448,A -85,B 0,C 180,E1 -20583.652,E2 -20583.652} C_VEL
LIN {X 0,Y 217.888,Z 675.745,A -85,B 0,C 180,E1 -20587.227,E2 -20587.227} C_VEL
LIN {X 0,Y 215.077,Z 681.585,A -85,B 0,C 180,E1 -20590.927,E2 -20590.927} C_VEL
LIN {X 0,Y 213.134,Z 686.128,A -85,B 0,C 180,E1 -20594.704,E2 -20594.704} C_VEL
LIN {X 0,Y 211.964,Z 689.456,A -85,B 0,C 180,E1 -20598.524,E2 -20598.524} C_VEL
LIN {X 0,Y 211.593,Z 691.612,A -85,B 0,C 180,E1 -20602.364,E2 -20602.364} C_VEL
LIN {X 0,Y 211.662,Z 692.55,A -85,B 0,C 180,E1 -20606.191,E2 -20606.191} C_VEL
LIN {X 0,Y 211.776,Z 692.578,A -85,B 0,C 180,E1 -20608.097,E2 -20608.097} C_VEL
LIN {X 0,Y 211.85,Z 692.302,A -85,B 0,C 180,E1 -20609.999,E2 -20609.999} C_VEL
LIN {X 0,Y 211.801,Z 691.712,A -85,B 0,C 180,E1 -20611.901,E2 -20611.901} C_VEL
LIN {X 0,Y 211.695,Z 689.583,A -85,B 0,C 180,E1 -20615.715,E2 -20615.715} C_VEL
LIN {X 0,Y 211.795,Z 686.144,A -85,B 0,C 180,E1 -20619.55,E2 -20619.55} C_VEL
LIN {X 0,Y 212.45,Z 681.317,A -85,B 0,C 180,E1 -20623.388,E2 -20623.388} C_VEL
LIN {X 0,Y 213.84,Z 674.977,A -85,B 0,C 180,E1 -20627.204,E2 -20627.204} C_VEL
LIN {X 0,Y 215.672,Z 668.066,A -85,B 0,C 180,E1 -20630.505,E2 -20630.505} C_VEL
LIN {X 0,Y 218.23,Z 659.694,A -85,B 0,C 180,E1 -20633.737,E2 -20633.737} C_VEL
LIN {X 0,Y 221.083,Z 649.94,A -85,B 0,C 180,E1 -20636.814,E2 -20636.814} C_VEL
LIN {X 0,Y 224.406,Z 639.218,A -85,B 0,C 180,E1 -20639.554,E2 -20639.554} C_VEL
LIN {X 0,Y 228.055,Z 626.888,A -85,B 0,C 180,E1 -20642.112,E2 -20642.112} C_VEL
LIN {X 0,Y 231.588,Z 614.575,A -85,B 0,C 180,E1 -20644.153,E2 -20644.153} C_VEL
LIN {X 0,Y 235.008,Z 600.762,A -85,B 0,C 180,E1 -20646.006,E2 -20646.006} C_VEL
LIN {X 0,Y 238.048,Z 586.499,A -85,B 0,C 180,E1 -20647.511,E2 -20647.511} C_VEL
LIN {X 0,Y 240.857,Z 571.256,A -85,B 0,C 180,E1 -20648.72,E2 -20648.72} C_VEL
LIN {X 0,Y 243.028,Z 555.175,A -85,B 0,C 180,E1 -20649.643,E2 -20649.643} C_VEL
LIN {X 0,Y 244.336,Z 539.088,A -85,B 0,C 180,E1 -20650.261,E2 -20650.261} C_VEL
LIN {X 0,Y 249.519,Z 454.684,A -85,B 0,C 180,E1 -20652.796,E2 -20652.796} C_VEL
LIN {X 0,Y 248.434,Z 445.926,A -85,B 0,C 180,E1 -20653.332,E2 -20653.332} C_VEL
LIN {X 0,Y 240.153,Z 426.319,A -85,B 0,C 180,E1 -20655.605,E2 -20655.605} C_VEL
LIN {X 0,Y 233.285,Z 411.657,A -85,B 0,C 180,E1 -20657.591,E2 -20657.591} C_VEL
LIN {X 0,Y 226.235,Z 397.966,A -85,B 0,C 180,E1 -20659.717,E2 -20659.717} C_VEL
LIN {X 0,Y 220.174,Z 387.137,A -85,B 0,C 180,E1 -20661.648,E2 -20661.648} C_VEL
LIN {X 0,Y 215.397,Z 378.74,A -85,B 0,C 180,E1 -20663.309,E2 -20663.309} C_VEL
LIN {X 0,Y 213.758,Z 373.472,A -85,B 0,C 180,E1 -20665.875,E2 -20665.875} C_VEL
LIN {X 0,Y 213.778,Z 373.481,A -85,B 0,C 180,E1 -20670.454,E2 -20670.454} C_VEL
LIN {X 0,Y 213.798,Z 373.474,A -85,B 0,C 180,E1 -20674.702,E2 -20674.702} C_VEL
LIN {X 0,Y 213.81,Z 373.475,A -85,B 0,C 180,E1 -20678.804,E2 -20678.804} C_VEL
LIN {X 0,Y 213.941,Z 373.457,A -85,B 0,C 180,E1 -20682.804,E2 -20682.804} C_VEL
LIN {X 0,Y 213.952,Z 373.441,A -85,B 0,C 180,E1 -20686.707,E2 -20686.707} C_VEL
LIN {X 0,Y 214.164,Z 373.401,A -85,B 0,C 180,E1 -20690.557,E2 -20690.557} C_VEL
LIN {X 0,Y 214.224,Z 373.416,A -85,B 0,C 180,E1 -20692.46,E2 -20692.46} C_VEL
LIN {X 0,Y 214.444,Z 373.376,A -85,B 0,C 180,E1 -20698.123,E2 -20698.123} C_VEL
LIN {X 0,Y 214.548,Z 373.37,A -85,B 0,C 180,E1 -20700.001,E2 -20700.001} C_VEL
LIN {X 0,Y 214.444,Z 373.396,A -85,B 0,C 180,E1 -20701.879,E2 -20701.879} C_VEL
LIN {X 0,Y 214.233,Z 373.399,A -85,B 0,C 180,E1 -20707.541,E2 -20707.541} C_VEL
LIN {X 0,Y 214.046,Z 373.448,A -85,B 0,C 180,E1 -20711.363,E2 -20711.363} C_VEL
LIN {X 0,Y 213.932,Z 373.44,A -85,B 0,C 180,E1 -20715.238,E2 -20715.238} C_VEL
LIN {X 0,Y 213.835,Z 373.466,A -85,B 0,C 180,E1 -20719.189,E2 -20719.189} C_VEL
LIN {X 0,Y 213.81,Z 373.468,A -85,B 0,C 180,E1 -20723.232,E2 -20723.232} C_VEL
LIN {X 0,Y 213.828,Z 373.457,A -85,B 0,C 180,E1 -20727.451,E2 -20727.451} C_VEL
LIN {X 0,Y 213.776,Z 373.478,A -85,B 0,C 180,E1 -20731.737,E2 -20731.737} C_VEL
LIN {X 0,Y 213.743,Z 373.467,A -85,B 0,C 180,E1 -20736.289,E2 -20736.289} C_VEL
LIN {X 0,Y 213.71,Z 373.483,A -85,B 0,C 180,E1 -20741.127,E2 -20741.127} C_VEL
LIN {X 0,Y 213.703,Z 373.466,A -85,B 0,C 180,E1 -20743.681,E2 -20743.681} C_VEL
LIN {X 0,Y 213.703,Z 373.487,A -85,B 0,C 180,E1 -20746.346,E2 -20746.346} C_VEL
LIN {X 0,Y 213.717,Z 373.483,A -85,B 0,C 180,E1 -20749.144,E2 -20749.144} C_VEL
LIN {X 0,Y 213.745,Z 373.483,A -85,B 0,C 180,E1 -20753.713,E2 -20753.713} C_VEL
LIN {X 0,Y 213.76,Z 373.468,A -85,B 0,C 180,E1 -20758.262,E2 -20758.262} C_VEL
LIN {X 0,Y 213.791,Z 373.475,A -85,B 0,C 180,E1 -20762.599,E2 -20762.599} C_VEL
LIN {X 0,Y 213.813,Z 373.477,A -85,B 0,C 180,E1 -20766.98,E2 -20766.98} C_VEL
LIN {X 0,Y 213.884,Z 373.466,A -85,B 0,C 180,E1 -20772.8,E2 -20772.8} C_VEL
LIN {X 0,Y 213.937,Z 373.465,A -85,B 0,C 180,E1 -20777.189,E2 -20777.189} C_VEL
LIN {X 0,Y 214.903,Z 376.191,A -85,B 0,C 180,E1 -20777.586,E2 -20777.586} C_VEL
LIN {X 0,Y 217.185,Z 378.976,A -85,B 0,C 180,E1 -20778.31,E2 -20778.31} C_VEL
LIN {X 0,Y 219.287,Z 382.101,A -85,B 0,C 180,E1 -20778.985,E2 -20778.985} C_VEL
LIN {X 0,Y 225.619,Z 391.627,A -85,B 0,C 180,E1 -20780.942,E2 -20780.942} C_VEL
LIN {X 0,Y 236.285,Z 408.879,A -85,B 0,C 180,E1 -20783.969,E2 -20783.969} C_VEL
LIN {X 0,Y 242.256,Z 420.126,A -85,B 0,C 180,E1 -20785.596,E2 -20785.596} C_VEL
LIN {X 0,Y 249.875,Z 434.959,A -85,B 0,C 180,E1 -20787.534,E2 -20787.534} C_VEL
LIN {X 0,Y 244.595,Z 522.375,A -85,B 0,C 180,E1 -20790.207,E2 -20790.207} C_VEL
LIN {X 0,Y 243.071,Z 537.582,A -85,B 0,C 180,E1 -20790.933,E2 -20790.933} C_VEL
LIN {X 0,Y 241.14,Z 552.324,A -85,B 0,C 180,E1 -20791.953,E2 -20791.953} C_VEL
LIN {X 0,Y 238.408,Z 567.958,A -85,B 0,C 180,E1 -20793.381,E2 -20793.381} C_VEL
LIN {X 0,Y 235.303,Z 582.688,A -85,B 0,C 180,E1 -20795.142,E2 -20795.142} C_VEL
LIN {X 0,Y 231.978,Z 596.228,A -85,B 0,C 180,E1 -20797.18,E2 -20797.18} C_VEL
LIN {X 0,Y 228.625,Z 608.417,A -85,B 0,C 180,E1 -20799.446,E2 -20799.446} C_VEL
LIN {X 0,Y 225.113,Z 620.265,A -85,B 0,C 180,E1 -20802.166,E2 -20802.166} C_VEL
LIN {X 0,Y 222.322,Z 629.225,A -85,B 0,C 180,E1 -20804.65,E2 -20804.65} C_VEL
LIN {X 0,Y 219.392,Z 638.339,A -85,B 0,C 180,E1 -20807.717,E2 -20807.717} C_VEL
LIN {X 0,Y 217.027,Z 645.955,A -85,B 0,C 180,E1 -20810.869,E2 -20810.869} C_VEL
LIN {X 0,Y 214.868,Z 652.966,A -85,B 0,C 180,E1 -20814.455,E2 -20814.455} C_VEL
LIN {X 0,Y 213.245,Z 659.144,A -85,B 0,C 180,E1 -20818.548,E2 -20818.548} C_VEL
LIN {X 0,Y 212.244,Z 663.023,A -85,B 0,C 180,E1 -20821.993,E2 -20821.993} C_VEL
LIN {X 0,Y 211.727,Z 665.089,A -85,B 0,C 180,E1 -20824.354,E2 -20824.354} C_VEL
LIN {X 0,Y 211.425,Z 666.904,A -85,B 0,C 180,E1 -20827.079,E2 -20827.079} C_VEL
LIN {X 0,Y 211.399,Z 668.148,A -85,B 0,C 180,E1 -20830.124,E2 -20830.124} C_VEL
LIN {X 0,Y 211.727,Z 668.727,A -85,B 0,C 180,E1 -20834.193,E2 -20834.193} C_VEL
LIN {X 0,Y 212.208,Z 668.424,A -85,B 0,C 180,E1 -20836.771,E2 -20836.771} C_VEL
LIN {X 0,Y 212.946,Z 667.603,A -85,B 0,C 180,E1 -20839.385,E2 -20839.385} C_VEL
LIN {X 0,Y 213.951,Z 666.187,A -85,B 0,C 180,E1 -20842.034,E2 -20842.034} C_VEL
LIN {X 0,Y 215.293,Z 664.141,A -85,B 0,C 180,E1 -20844.697,E2 -20844.697} C_VEL
LIN {X 0,Y 216.987,Z 661.485,A -85,B 0,C 180,E1 -20847.365,E2 -20847.365} C_VEL
LIN {X 0,Y 220.362,Z 656.051,A -85,B 0,C 180,E1 -20851.419,E2 -20851.419} C_VEL
LIN {X 0,Y 224.485,Z 649.14,A -85,B 0,C 180,E1 -20855.22,E2 -20855.22} C_VEL
LIN {X 0,Y 228.703,Z 641.731,A -85,B 0,C 180,E1 -20858.36,E2 -20858.36} C_VEL
LIN {X 0,Y 233.068,Z 633.711,A -85,B 0,C 180,E1 -20861.085,E2 -20861.085} C_VEL
LIN {X 0,Y 237.656,Z 624.42,A -85,B 0,C 180,E1 -20863.683,E2 -20863.683} C_VEL
LIN {X 0,Y 242.488,Z 613.95,A -85,B 0,C 180,E1 -20866.037,E2 -20866.037} C_VEL
LIN {X 0,Y 247.312,Z 602.447,A -85,B 0,C 180,E1 -20868.13,E2 -20868.13} C_VEL
LIN {X 0,Y 251.685,Z 590.652,A -85,B 0,C 180,E1 -20869.886,E2 -20869.886} C_VEL
LIN {X 0,Y 255.842,Z 577.56,A -85,B 0,C 180,E1 -20871.468,E2 -20871.468} C_VEL
LIN {X 0,Y 259.585,Z 563.602,A -85,B 0,C 180,E1 -20872.787,E2 -20872.787} C_VEL
LIN {X 0,Y 262.718,Z 548.707,A -85,B 0,C 180,E1 -20873.881,E2 -20873.881} C_VEL
LIN {X 0,Y 265.11,Z 533.471,A -85,B 0,C 180,E1 -20874.699,E2 -20874.699} C_VEL
LIN {X 0,Y 266.947,Z 516.638,A -85,B 0,C 180,E1 -20875.28,E2 -20875.28} C_VEL
LIN {X 0,Y 272.841,Z 448.994,A -85,B 0,C 180,E1 -20877.253,E2 -20877.253} C_VEL
LIN {X 0,Y 268.113,Z 439.639,A -85,B 0,C 180,E1 -20879.59,E2 -20879.59} C_VEL
LIN {X 0,Y 265.054,Z 434.501,A -85,B 0,C 180,E1 -20881.224,E2 -20881.224} C_VEL
LIN {X 0,Y 260.995,Z 427.349,A -85,B 0,C 180,E1 -20883.775,E2 -20883.775} C_VEL
LIN {X 0,Y 258.573,Z 423.734,A -85,B 0,C 180,E1 -20885.503,E2 -20885.503} C_VEL
LIN {X 0,Y 255.693,Z 419.651,A -85,B 0,C 180,E1 -20887.899,E2 -20887.899} C_VEL
LIN {X 0,Y 253.374,Z 416.455,A -85,B 0,C 180,E1 -20890.275,E2 -20890.275} C_VEL
LIN {X 0,Y 252.83,Z 415.318,A -85,B 0,C 180,E1 -20891.03,E2 -20891.03} C_VEL
LIN {X 0,Y 250.431,Z 413.038,A -85,B 0,C 180,E1 -20894.81,E2 -20894.81} C_VEL
LIN {X 0,Y 249.757,Z 410.883,A -85,B 0,C 180,E1 -20897.61,E2 -20897.61} C_VEL
LIN {X 0,Y 249.565,Z 410.998,A -85,B 0,C 180,E1 -20898.705,E2 -20898.705} C_VEL
LIN {X 0,Y 249.391,Z 411.961,A -85,B 0,C 180,E1 -20900.043,E2 -20900.043} C_VEL
LIN {X 0,Y 249.245,Z 414.005,A -85,B 0,C 180,E1 -20901.328,E2 -20901.328} C_VEL
LIN {X 0,Y 249.452,Z 420.708,A -85,B 0,C 180,E1 -20904.683,E2 -20904.683} C_VEL
LIN {X 0,Y 249.8,Z 421.834,A -85,B 0,C 180,E1 -20905.563,E2 -20905.563} C_VEL
LIN {X 0,Y 252.595,Z 426.918,A -85,B 0,C 180,E1 -20909.628,E2 -20909.628} C_VEL
LIN {X 0,Y 255.548,Z 432.801,A -85,B 0,C 180,E1 -20912.628,E2 -20912.628} C_VEL
LIN {X 0,Y 258.5,Z 438.988,A -85,B 0,C 180,E1 -20915.039,E2 -20915.039} C_VEL
LIN {X 0,Y 261.566,Z 445.671,A -85,B 0,C 180,E1 -20917.152,E2 -20917.152} C_VEL
LIN {X 0,Y 265.039,Z 454.118,A -85,B 0,C 180,E1 -20919.297,E2 -20919.297} C_VEL
LIN {X 0,Y 268.239,Z 463.141,A -85,B 0,C 180,E1 -20921.135,E2 -20921.135} C_VEL
LIN {X 0,Y 263.239,Z 518.24,A -85,B 0,C 180,E1 -20922.73,E2 -20922.73} C_VEL
LIN {X 0,Y 260.572,Z 545.195,A -85,B 0,C 180,E1 -20923.542,E2 -20923.542} C_VEL
LIN {X 0,Y 258.019,Z 560.643,A -85,B 0,C 180,E1 -20924.216,E2 -20924.216} C_VEL
LIN {X 0,Y 254.558,Z 575.717,A -85,B 0,C 180,E1 -20925.109,E2 -20925.109} C_VEL
LIN {X 0,Y 250.402,Z 590.349,A -85,B 0,C 180,E1 -20926.278,E2 -20926.278} C_VEL
LIN {X 0,Y 245.578,Z 604.494,A -85,B 0,C 180,E1 -20927.737,E2 -20927.737} C_VEL
LIN {X 0,Y 240.596,Z 617.421,A -85,B 0,C 180,E1 -20929.462,E2 -20929.462} C_VEL
LIN {X 0,Y 235.865,Z 628.393,A -85,B 0,C 180,E1 -20931.263,E2 -20931.263} C_VEL
LIN {X 0,Y 230.592,Z 639.547,A -85,B 0,C 180,E1 -20933.535,E2 -20933.535} C_VEL
LIN {X 0,Y 224.951,Z 650.577,A -85,B 0,C 180,E1 -20936.319,E2 -20936.319} C_VEL
LIN {X 0,Y 220.045,Z 659.809,A -85,B 0,C 180,E1 -20939.267,E2 -20939.267} C_VEL
LIN {X 0,Y 215.306,Z 668.596,A -85,B 0,C 180,E1 -20942.806,E2 -20942.806} C_VEL
LIN {X 0,Y 211.305,Z 675.761,A -85,B 0,C 180,E1 -20946.476,E2 -20946.476} C_VEL
LIN {X 0,Y 208.324,Z 681.502,A -85,B 0,C 180,E1 -20950.283,E2 -20950.283} C_VEL
LIN {X 0,Y 206.213,Z 685.942,A -85,B 0,C 180,E1 -20954.177,E2 -20954.177} C_VEL
LIN {X 0,Y 204.936,Z 689.172,A -85,B 0,C 180,E1 -20958.125,E2 -20958.125} C_VEL
LIN {X 0,Y 204.514,Z 691.256,A -85,B 0,C 180,E1 -20962.098,E2 -20962.098} C_VEL
LIN {X 0,Y 204.567,Z 692.152,A -85,B 0,C 180,E1 -20966.059,E2 -20966.059} C_VEL
LIN {X 0,Y 204.704,Z 692.142,A -85,B 0,C 180,E1 -20968.032,E2 -20968.032} C_VEL
LIN {X 0,Y 204.779,Z 691.827,A -85,B 0,C 180,E1 -20969.999,E2 -20969.999} C_VEL
LIN {X 0,Y 204.73,Z 691.199,A -85,B 0,C 180,E1 -20971.966,E2 -20971.966} C_VEL
LIN {X 0,Y 204.588,Z 688.989,A -85,B 0,C 180,E1 -20975.914,E2 -20975.914} C_VEL
LIN {X 0,Y 204.748,Z 685.469,A -85,B 0,C 180,E1 -20979.881,E2 -20979.881} C_VEL
LIN {X 0,Y 205.481,Z 680.552,A -85,B 0,C 180,E1 -20983.851,E2 -20983.851} C_VEL
LIN {X 0,Y 206.982,Z 674.113,A -85,B 0,C 180,E1 -20987.793,E2 -20987.793} C_VEL
LIN {X 0,Y 209.265,Z 665.968,A -85,B 0,C 180,E1 -20991.679,E2 -20991.679} C_VEL
LIN {X 0,Y 212.061,Z 657.265,A -85,B 0,C 180,E1 -20994.995,E2 -20994.995} C_VEL
LIN {X 0,Y 215.18,Z 647.119,A -85,B 0,C 180,E1 -20998.135,E2 -20998.135} C_VEL
LIN {X 0,Y 218.748,Z 635.905,A -85,B 0,C 180,E1 -21000.933,E2 -21000.933} C_VEL
LIN {X 0,Y 222.343,Z 624.147,A -85,B 0,C 180,E1 -21003.311,E2 -21003.311} C_VEL
LIN {X 0,Y 225.96,Z 611.354,A -85,B 0,C 180,E1 -21005.4,E2 -21005.4} C_VEL
LIN {X 0,Y 228.985,Z 599.537,A -85,B 0,C 180,E1 -21006.967,E2 -21006.967} C_VEL
LIN {X 0,Y 232.154,Z 585.032,A -85,B 0,C 180,E1 -21008.497,E2 -21008.497} C_VEL
LIN {X 0,Y 235.054,Z 569.38,A -85,B 0,C 180,E1 -21009.724,E2 -21009.724} C_VEL
LIN {X 0,Y 237.064,Z 554.701,A -85,B 0,C 180,E1 -21010.568,E2 -21010.568} C_VEL
LIN {X 0,Y 238.417,Z 538.624,A -85,B 0,C 180,E1 -21011.195,E2 -21011.195} C_VEL
LIN {X 0,Y 243.738,Z 454.878,A -85,B 0,C 180,E1 -21013.762,E2 -21013.762} C_VEL
LIN {X 0,Y 242.775,Z 448.32,A -85,B 0,C 180,E1 -21014.199,E2 -21014.199} C_VEL
LIN {X 0,Y 234.057,Z 427.666,A -85,B 0,C 180,E1 -21016.711,E2 -21016.711} C_VEL
LIN {X 0,Y 226.477,Z 411.687,A -85,B 0,C 180,E1 -21019.003,E2 -21019.003} C_VEL
LIN {X 0,Y 218.972,Z 397.374,A -85,B 0,C 180,E1 -21021.414,E2 -21021.414} C_VEL
LIN {X 0,Y 212.912,Z 386.772,A -85,B 0,C 180,E1 -21023.474,E2 -21023.474} C_VEL
LIN {X 0,Y 207.872,Z 378.191,A -85,B 0,C 180,E1 -21025.361,E2 -21025.361} C_VEL
LIN {X 0,Y 206.699,Z 374.35,A -85,B 0,C 180,E1 -21027.376,E2 -21027.376} C_VEL
LIN {X 0,Y 206.763,Z 374.357,A -85,B 0,C 180,E1 -21032.097,E2 -21032.097} C_VEL
LIN {X 0,Y 206.783,Z 374.351,A -85,B 0,C 180,E1 -21036.584,E2 -21036.584} C_VEL
LIN {X 0,Y 206.871,Z 374.335,A -85,B 0,C 180,E1 -21042.197,E2 -21042.197} C_VEL
LIN {X 0,Y 206.894,Z 374.325,A -85,B 0,C 180,E1 -21046.245,E2 -21046.245} C_VEL
LIN {X 0,Y 207.103,Z 374.275,A -85,B 0,C 180,E1 -21050.232,E2 -21050.232} C_VEL
LIN {X 0,Y 207.165,Z 374.292,A -85,B 0,C 180,E1 -21052.202,E2 -21052.202} C_VEL
LIN {X 0,Y 207.38,Z 374.255,A -85,B 0,C 180,E1 -21058.059,E2 -21058.059} C_VEL
LIN {X 0,Y 207.513,Z 374.245,A -85,B 0,C 180,E1 -21060.001,E2 -21060.001} C_VEL
LIN {X 0,Y 207.381,Z 374.276,A -85,B 0,C 180,E1 -21061.943,E2 -21061.943} C_VEL
LIN {X 0,Y 207.177,Z 374.278,A -85,B 0,C 180,E1 -21067.799,E2 -21067.799} C_VEL
LIN {X 0,Y 206.982,Z 374.327,A -85,B 0,C 180,E1 -21071.756,E2 -21071.756} C_VEL
LIN {X 0,Y 206.865,Z 374.315,A -85,B 0,C 180,E1 -21075.772,E2 -21075.772} C_VEL
LIN {X 0,Y 206.778,Z 374.349,A -85,B 0,C 180,E1 -21079.87,E2 -21079.87} C_VEL
LIN {X 0,Y 206.746,Z 374.338,A -85,B 0,C 180,E1 -21084.075,E2 -21084.075} C_VEL
LIN {X 0,Y 206.743,Z 374.348,A -85,B 0,C 180,E1 -21088.42,E2 -21088.42} C_VEL
LIN {X 0,Y 206.701,Z 374.349,A -85,B 0,C 180,E1 -21092.958,E2 -21092.958} C_VEL
LIN {X 0,Y 206.68,Z 374.36,A -85,B 0,C 180,E1 -21097.741,E2 -21097.741} C_VEL
LIN {X 0,Y 206.64,Z 374.36,A -85,B 0,C 180,E1 -21101.564,E2 -21101.564} C_VEL
LIN {X 0,Y 206.631,Z 374.362,A -85,B 0,C 180,E1 -21105.584,E2 -21105.584} C_VEL
LIN {X 0,Y 206.66,Z 374.356,A -85,B 0,C 180,E1 -21109.75,E2 -21109.75} C_VEL
LIN {X 0,Y 206.7,Z 374.366,A -85,B 0,C 180,E1 -21114.69,E2 -21114.69} C_VEL
LIN {X 0,Y 206.697,Z 374.351,A -85,B 0,C 180,E1 -21119.336,E2 -21119.336} C_VEL
LIN {X 0,Y 206.707,Z 374.349,A -85,B 0,C 180,E1 -21123.77,E2 -21123.77} C_VEL
LIN {X 0,Y 206.733,Z 374.354,A -85,B 0,C 180,E1 -21128.042,E2 -21128.042} C_VEL
LIN {X 0,Y 206.824,Z 374.349,A -85,B 0,C 180,E1 -21132.193,E2 -21132.193} C_VEL
LIN {X 0,Y 206.835,Z 374.438,A -85,B 0,C 180,E1 -21135.301,E2 -21135.301} C_VEL
LIN {X 0,Y 207.824,Z 377.188,A -85,B 0,C 180,E1 -21135.733,E2 -21135.733} C_VEL
LIN {X 0,Y 210.112,Z 379.842,A -85,B 0,C 180,E1 -21136.518,E2 -21136.518} C_VEL
LIN {X 0,Y 212.238,Z 383.065,A -85,B 0,C 180,E1 -21137.265,E2 -21137.265} C_VEL
LIN {X 0,Y 214.092,Z 385.783,A -85,B 0,C 180,E1 -21137.891,E2 -21137.891} C_VEL
LIN {X 0,Y 218.658,Z 392.289,A -85,B 0,C 180,E1 -21139.355,E2 -21139.355} C_VEL
LIN {X 0,Y 231.595,Z 413.277,A -85,B 0,C 180,E1 -21143.234,E2 -21143.234} C_VEL
LIN {X 0,Y 237.421,Z 424.393,A -85,B 0,C 180,E1 -21144.877,E2 -21144.877} C_VEL
LIN {X 0,Y 244.067,Z 437.327,A -85,B 0,C 180,E1 -21146.641,E2 -21146.641} C_VEL
LIN {X 0,Y 238.615,Z 523.27,A -85,B 0,C 180,E1 -21149.316,E2 -21149.316} C_VEL
LIN {X 0,Y 236.948,Z 539.141,A -85,B 0,C 180,E1 -21150.107,E2 -21150.107} C_VEL
LIN {X 0,Y 234.885,Z 554,A -85,B 0,C 180,E1 -21151.179,E2 -21151.179} C_VEL
LIN {X 0,Y 232.162,Z 568.747,A -85,B 0,C 180,E1 -21152.575,E2 -21152.575} C_VEL
LIN {X 0,Y 229.32,Z 581.951,A -85,B 0,C 180,E1 -21154.175,E2 -21154.175} C_VEL
LIN {X 0,Y 225.963,Z 595.351,A -85,B 0,C 180,E1 -21156.192,E2 -21156.192} C_VEL
LIN {X 0,Y 222.248,Z 608.397,A -85,B 0,C 180,E1 -21158.64,E2 -21158.64} C_VEL
LIN {X 0,Y 219.04,Z 619.052,A -85,B 0,C 180,E1 -21161.1,E2 -21161.1} C_VEL
LIN {X 0,Y 215.624,Z 629.567,A -85,B 0,C 180,E1 -21164.054,E2 -21164.054} C_VEL
LIN {X 0,Y 212.502,Z 638.978,A -85,B 0,C 180,E1 -21167.318,E2 -21167.318} C_VEL
LIN {X 0,Y 209.724,Z 647.504,A -85,B 0,C 180,E1 -21171.009,E2 -21171.009} C_VEL
LIN {X 0,Y 207.889,Z 653.253,A -85,B 0,C 180,E1 -21174.106,E2 -21174.106} C_VEL
LIN {X 0,Y 206.408,Z 658.642,A -85,B 0,C 180,E1 -21177.713,E2 -21177.713} C_VEL
LIN {X 0,Y 205.339,Z 662.674,A -85,B 0,C 180,E1 -21181.166,E2 -21181.166} C_VEL
LIN {X 0,Y 204.616,Z 665.562,A -85,B 0,C 180,E1 -21184.477,E2 -21184.477} C_VEL
LIN {X 0,Y 204.271,Z 667.794,A -85,B 0,C 180,E1 -21188.266,E2 -21188.266} C_VEL
LIN {X 0,Y 204.326,Z 668.704,A -85,B 0,C 180,E1 -21190.824,E2 -21190.824} C_VEL
LIN {X 0,Y 204.591,Z 669.181,A -85,B 0,C 180,E1 -21193.83,E2 -21193.83} C_VEL
LIN {X 0,Y 205.103,Z 668.956,A -85,B 0,C 180,E1 -21196.739,E2 -21196.739} C_VEL
LIN {X 0,Y 205.902,Z 668.179,A -85,B 0,C 180,E1 -21199.569,E2 -21199.569} C_VEL
LIN {X 0,Y 206.982,Z 666.873,A -85,B 0,C 180,E1 -21202.324,E2 -21202.324} C_VEL
LIN {X 0,Y 208.355,Z 664.971,A -85,B 0,C 180,E1 -21205.01,E2 -21205.01} C_VEL
LIN {X 0,Y 210.886,Z 661.329,A -85,B 0,C 180,E1 -21208.759,E2 -21208.759} C_VEL
LIN {X 0,Y 214.374,Z 656.029,A -85,B 0,C 180,E1 -21212.678,E2 -21212.678} C_VEL
LIN {X 0,Y 218.502,Z 649.546,A -85,B 0,C 180,E1 -21216.292,E2 -21216.292} C_VEL
LIN {X 0,Y 223.393,Z 641.475,A -85,B 0,C 180,E1 -21219.753,E2 -21219.753} C_VEL
LIN {X 0,Y 228.604,Z 632.198,A -85,B 0,C 180,E1 -21222.863,E2 -21222.863} C_VEL
LIN {X 0,Y 233.852,Z 621.955,A -85,B 0,C 180,E1 -21225.615,E2 -21225.615} C_VEL
LIN {X 0,Y 238.827,Z 611.482,A -85,B 0,C 180,E1 -21227.862,E2 -21227.862} C_VEL
LIN {X 0,Y 243.544,Z 600.441,A -85,B 0,C 180,E1 -21229.777,E2 -21229.777} C_VEL
LIN {X 0,Y 248.593,Z 586.864,A -85,B 0,C 180,E1 -21231.689,E2 -21231.689} C_VEL
LIN {X 0,Y 252.839,Z 573.266,A -85,B 0,C 180,E1 -21233.215,E2 -21233.215} C_VEL
LIN {X 0,Y 256.7,Z 558.447,A -85,B 0,C 180,E1 -21234.501,E2 -21234.501} C_VEL
LIN {X 0,Y 259.655,Z 543.577,A -85,B 0,C 180,E1 -21235.49,E2 -21235.49} C_VEL
LIN {X 0,Y 261.799,Z 529.048,A -85,B 0,C 180,E1 -21236.168,E2 -21236.168} C_VEL
LIN {X 0,Y 268.271,Z 459.587,A -85,B 0,C 180,E1 -21238.217,E2 -21238.217} C_VEL
LIN {X 0,Y 268.866,Z 452.406,A -85,B 0,C 180,E1 -21238.452,E2 -21238.452} C_VEL
LIN {X 0,Y 264.396,Z 443.33,A -85,B 0,C 180,E1 -21240.875,E2 -21240.875} C_VEL
LIN {X 0,Y 259.034,Z 433.795,A -85,B 0,C 180,E1 -21244.278,E2 -21244.278} C_VEL
LIN {X 0,Y 256.747,Z 430.234,A -85,B 0,C 180,E1 -21246.004,E2 -21246.004} C_VEL
LIN {X 0,Y 254.146,Z 426.362,A -85,B 0,C 180,E1 -21248.292,E2 -21248.292} C_VEL
LIN {X 0,Y 251.878,Z 423.026,A -85,B 0,C 180,E1 -21250.781,E2 -21250.781} C_VEL
LIN {X 0,Y 251.546,Z 422.224,A -85,B 0,C 180,E1 -21251.278,E2 -21251.278} C_VEL
LIN {X 0,Y 249.258,Z 419.957,A -85,B 0,C 180,E1 -21255.064,E2 -21255.064} C_VEL
LIN {X 0,Y 248.728,Z 418.103,A -85,B 0,C 180,E1 -21257.326,E2 -21257.326} C_VEL
LIN {X 0,Y 248.445,Z 418.113,A -85,B 0,C 180,E1 -21259.184,E2 -21259.184} C_VEL
LIN {X 0,Y 249.223,Z 420.065,A -85,B 0,C 180,E1 -21264.043,E2 -21264.043} C_VEL
LIN {X 0,Y 249.8,Z 421.834,A -85,B 0,C 180,E1 -21265.563,E2 -21265.563} C_VEL
LIN {X 0,Y 250.412,Z 423.879,A -85,B 0,C 180,E1 -21266.822,E2 -21266.822} C_VEL
LIN {X 0,Y 250.926,Z 426.981,A -85,B 0,C 180,E1 -21267.976,E2 -21267.976} C_VEL
LIN {X 0,Y 252.067,Z 434.251,A -85,B 0,C 180,E1 -21270.153,E2 -21270.153} C_VEL
LIN {X 0,Y 252.972,Z 437.438,A -85,B 0,C 180,E1 -21271.293,E2 -21271.293} C_VEL
LIN {X 0,Y 253.356,Z 438.304,A -85,B 0,C 180,E1 -21271.693,E2 -21271.693} C_VEL
LIN {X 0,Y 256.353,Z 445.011,A -85,B 0,C 180,E1 -21274.349,E2 -21274.349} C_VEL
LIN {X 0,Y 259.234,Z 451.713,A -85,B 0,C 180,E1 -21276.489,E2 -21276.489} C_VEL
LIN {X 0,Y 262.406,Z 459.963,A -85,B 0,C 180,E1 -21278.604,E2 -21278.604} C_VEL
LIN {X 0,Y 264.53,Z 466.254,A -85,B 0,C 180,E1 -21279.921,E2 -21279.921} C_VEL
LIN {X 0,Y 256.978,Z 543.183,A -85,B 0,C 180,E1 -21282.139,E2 -21282.139} C_VEL
LIN {X 0,Y 254.415,Z 558.802,A -85,B 0,C 180,E1 -21282.796,E2 -21282.796} C_VEL
LIN {X 0,Y 250.869,Z 574.187,A -85,B 0,C 180,E1 -21283.686,E2 -21283.686} C_VEL
LIN {X 0,Y 246.575,Z 588.993,A -85,B 0,C 180,E1 -21284.845,E2 -21284.845} C_VEL
LIN {X 0,Y 241.534,Z 603.234,A -85,B 0,C 180,E1 -21286.285,E2 -21286.285} C_VEL
LIN {X 0,Y 236.584,Z 615.636,A -85,B 0,C 180,E1 -21287.91,E2 -21287.91} C_VEL
LIN {X 0,Y 231.333,Z 627.338,A -85,B 0,C 180,E1 -21289.807,E2 -21289.807} C_VEL
LIN {X 0,Y 225.804,Z 638.536,A -85,B 0,C 180,E1 -21292.069,E2 -21292.069} C_VEL
LIN {X 0,Y 219.887,Z 649.606,A -85,B 0,C 180,E1 -21294.877,E2 -21294.877} C_VEL
LIN {X 0,Y 214.615,Z 658.88,A -85,B 0,C 180,E1 -21297.849,E2 -21297.849} C_VEL
LIN {X 0,Y 209.541,Z 667.755,A -85,B 0,C 180,E1 -21301.448,E2 -21301.448} C_VEL
LIN {X 0,Y 205.69,Z 674.147,A -85,B 0,C 180,E1 -21304.715,E2 -21304.715} C_VEL
LIN {X 0,Y 202.281,Z 680.116,A -85,B 0,C 180,E1 -21308.603,E2 -21308.603} C_VEL
LIN {X 0,Y 199.832,Z 684.801,A -85,B 0,C 180,E1 -21312.605,E2 -21312.605} C_VEL
LIN {X 0,Y 198.528,Z 687.483,A -85,B 0,C 180,E1 -21315.652,E2 -21315.652} C_VEL
LIN {X 0,Y 197.598,Z 690.043,A -85,B 0,C 180,E1 -21319.755,E2 -21319.755} C_VEL
LIN {X 0,Y 197.392,Z 691.467,A -85,B 0,C 180,E1 -21323.867,E2 -21323.867} C_VEL
LIN {X 0,Y 197.632,Z 691.707,A -85,B 0,C 180,E1 -21327.961,E2 -21327.961} C_VEL
LIN {X 0,Y 197.71,Z 691.353,A -85,B 0,C 180,E1 -21329.999,E2 -21329.999} C_VEL
LIN {X 0,Y 197.661,Z 690.683,A -85,B 0,C 180,E1 -21332.037,E2 -21332.037} C_VEL
LIN {X 0,Y 197.545,Z 689.159,A -85,B 0,C 180,E1 -21335.036,E2 -21335.036} C_VEL
LIN {X 0,Y 197.514,Z 686.745,A -85,B 0,C 180,E1 -21338.182,E2 -21338.182} C_VEL
LIN {X 0,Y 197.981,Z 682.443,A -85,B 0,C 180,E1 -21342.297,E2 -21342.297} C_VEL
LIN {X 0,Y 199.2,Z 676.681,A -85,B 0,C 180,E1 -21346.393,E2 -21346.393} C_VEL
LIN {X 0,Y 201.26,Z 669.309,A -85,B 0,C 180,E1 -21350.437,E2 -21350.437} C_VEL
LIN {X 0,Y 203.76,Z 661.37,A -85,B 0,C 180,E1 -21353.907,E2 -21353.907} C_VEL
LIN {X 0,Y 206.442,Z 653.303,A -85,B 0,C 180,E1 -21356.812,E2 -21356.812} C_VEL
LIN {X 0,Y 209.623,Z 643.578,A -85,B 0,C 180,E1 -21359.689,E2 -21359.689} C_VEL
LIN {X 0,Y 213.585,Z 631.424,A -85,B 0,C 180,E1 -21362.602,E2 -21362.602} C_VEL
LIN {X 0,Y 217.459,Z 618.85,A -85,B 0,C 180,E1 -21365.005,E2 -21365.005} C_VEL
LIN {X 0,Y 221.419,Z 605.011,A -85,B 0,C 180,E1 -21367.089,E2 -21367.089} C_VEL
LIN {X 0,Y 224.595,Z 591.4,A -85,B 0,C 180,E1 -21368.743,E2 -21368.743} C_VEL
LIN {X 0,Y 227.707,Z 576.53,A -85,B 0,C 180,E1 -21370.111,E2 -21370.111} C_VEL
LIN {X 0,Y 230.089,Z 561.953,A -85,B 0,C 180,E1 -21371.121,E2 -21371.121} C_VEL
LIN {X 0,Y 232.001,Z 546.291,A -85,B 0,C 180,E1 -21371.865,E2 -21371.865} C_VEL
LIN {X 0,Y 237.96,Z 456.44,A -85,B 0,C 180,E1 -21374.705,E2 -21374.705} C_VEL
LIN {X 0,Y 237.215,Z 451.019,A -85,B 0,C 180,E1 -21375.075,E2 -21375.075} C_VEL
LIN {X 0,Y 229.135,Z 431.591,A -85,B 0,C 180,E1 -21377.513,E2 -21377.513} C_VEL
LIN {X 0,Y 221.118,Z 414.643,A -85,B 0,C 180,E1 -21380.042,E2 -21380.042} C_VEL
LIN {X 0,Y 214.268,Z 401.464,A -85,B 0,C 180,E1 -21382.346,E2 -21382.346} C_VEL
LIN {X 0,Y 208.037,Z 390.432,A -85,B 0,C 180,E1 -21384.566,E2 -21384.566} C_VEL
LIN {X 0,Y 202.543,Z 381.424,A -85,B 0,C 180,E1 -21386.651,E2 -21386.651} C_VEL
LIN {X 0,Y 200.455,Z 377.695,A -85,B 0,C 180,E1 -21387.524,E2 -21387.524} C_VEL
LIN {X 0,Y 199.686,Z 375.239,A -85,B 0,C 180,E1 -21388.874,E2 -21388.874} C_VEL
LIN {X 0,Y 199.684,Z 375.238,A -85,B 0,C 180,E1 -21392.772,E2 -21392.772} C_VEL
LIN {X 0,Y 199.735,Z 375.224,A -85,B 0,C 180,E1 -21397.229,E2 -21397.229} C_VEL
LIN {X 0,Y 199.794,Z 375.216,A -85,B 0,C 180,E1 -21401.758,E2 -21401.758} C_VEL
LIN {X 0,Y 199.834,Z 375.21,A -85,B 0,C 180,E1 -21405.749,E2 -21405.749} C_VEL
LIN {X 0,Y 200.068,Z 375.146,A -85,B 0,C 180,E1 -21409.885,E2 -21409.885} C_VEL
LIN {X 0,Y 200.032,Z 375.192,A -85,B 0,C 180,E1 -21413.95,E2 -21413.95} C_VEL
LIN {X 0,Y 200.32,Z 375.133,A -85,B 0,C 180,E1 -21417.99,E2 -21417.99} C_VEL
LIN {X 0,Y 200.478,Z 375.12,A -85,B 0,C 180,E1 -21420.001,E2 -21420.001} C_VEL
LIN {X 0,Y 200.031,Z 375.191,A -85,B 0,C 180,E1 -21424.03,E2 -21424.03} C_VEL
LIN {X 0,Y 200.122,Z 375.157,A -85,B 0,C 180,E1 -21428.076,E2 -21428.076} C_VEL
LIN {X 0,Y 199.913,Z 375.208,A -85,B 0,C 180,E1 -21432.178,E2 -21432.178} C_VEL
LIN {X 0,Y 199.802,Z 375.192,A -85,B 0,C 180,E1 -21436.344,E2 -21436.344} C_VEL
LIN {X 0,Y 199.69,Z 375.235,A -85,B 0,C 180,E1 -21440.607,E2 -21440.607} C_VEL
LIN {X 0,Y 199.663,Z 375.21,A -85,B 0,C 180,E1 -21444.987,E2 -21444.987} C_VEL
LIN {X 0,Y 199.674,Z 375.236,A -85,B 0,C 180,E1 -21449.523,E2 -21449.523} C_VEL
LIN {X 0,Y 199.677,Z 375.228,A -85,B 0,C 180,E1 -21452.359,E2 -21452.359} C_VEL
LIN {X 0,Y 199.623,Z 375.228,A -85,B 0,C 180,E1 -21456.764,E2 -21456.764} C_VEL
LIN {X 0,Y 199.608,Z 375.246,A -85,B 0,C 180,E1 -21459.329,E2 -21459.329} C_VEL
LIN {X 0,Y 199.572,Z 375.23,A -85,B 0,C 180,E1 -21462.311,E2 -21462.311} C_VEL
LIN {X 0,Y 199.577,Z 375.235,A -85,B 0,C 180,E1 -21465.229,E2 -21465.229} C_VEL
LIN {X 0,Y 199.578,Z 375.251,A -85,B 0,C 180,E1 -21468.006,E2 -21468.006} C_VEL
LIN {X 0,Y 199.61,Z 375.225,A -85,B 0,C 180,E1 -21470.769,E2 -21470.769} C_VEL
LIN {X 0,Y 199.612,Z 375.246,A -85,B 0,C 180,E1 -21475.715,E2 -21475.715} C_VEL
LIN {X 0,Y 199.687,Z 375.219,A -85,B 0,C 180,E1 -21478.136,E2 -21478.136} C_VEL
LIN {X 0,Y 199.645,Z 375.235,A -85,B 0,C 180,E1 -21482.767,E2 -21482.767} C_VEL
LIN {X 0,Y 199.709,Z 375.234,A -85,B 0,C 180,E1 -21487.227,E2 -21487.227} C_VEL
LIN {X 0,Y 199.764,Z 375.22,A -85,B 0,C 180,E1 -21493.194,E2 -21493.194} C_VEL
LIN {X 0,Y 200.758,Z 378.061,A -85,B 0,C 180,E1 -21493.737,E2 -21493.737} C_VEL
LIN {X 0,Y 202.993,Z 380.606,A -85,B 0,C 180,E1 -21494.558,E2 -21494.558} C_VEL
LIN {X 0,Y 205.18,Z 384.003,A -85,B 0,C 180,E1 -21495.384,E2 -21495.384} C_VEL
LIN {X 0,Y 206.426,Z 385.539,A -85,B 0,C 180,E1 -21495.819,E2 -21495.819} C_VEL
LIN {X 0,Y 214.367,Z 397.084,A -85,B 0,C 180,E1 -21498.561,E2 -21498.561} C_VEL
LIN {X 0,Y 227.047,Z 417.877,A -85,B 0,C 180,E1 -21502.509,E2 -21502.509} C_VEL
LIN {X 0,Y 232.75,Z 428.873,A -85,B 0,C 180,E1 -21504.169,E2 -21504.169} C_VEL
LIN {X 0,Y 238.28,Z 439.796,A -85,B 0,C 180,E1 -21505.709,E2 -21505.709} C_VEL
LIN {X 0,Y 232.647,Z 524.363,A -85,B 0,C 180,E1 -21508.388,E2 -21508.388} C_VEL
LIN {X 0,Y 230.949,Z 540.007,A -85,B 0,C 180,E1 -21509.2,E2 -21509.2} C_VEL
LIN {X 0,Y 228.705,Z 555.223,A -85,B 0,C 180,E1 -21510.331,E2 -21510.331} C_VEL
LIN {X 0,Y 225.869,Z 570.017,A -85,B 0,C 180,E1 -21511.784,E2 -21511.784} C_VEL
LIN {X 0,Y 222.555,Z 584.509,A -85,B 0,C 180,E1 -21513.622,E2 -21513.622} C_VEL
LIN {X 0,Y 218.983,Z 597.985,A -85,B 0,C 180,E1 -21515.775,E2 -21515.775} C_VEL
LIN {X 0,Y 215.663,Z 609.165,A -85,B 0,C 180,E1 -21517.962,E2 -21517.962} C_VEL
LIN {X 0,Y 212.351,Z 619.781,A -85,B 0,C 180,E1 -21520.489,E2 -21520.489} C_VEL
LIN {X 0,Y 208.698,Z 630.574,A -85,B 0,C 180,E1 -21523.635,E2 -21523.635} C_VEL
LIN {X 0,Y 205.621,Z 639.528,A -85,B 0,C 180,E1 -21526.856,E2 -21526.856} C_VEL
LIN {X 0,Y 202.771,Z 647.97,A -85,B 0,C 180,E1 -21530.637,E2 -21530.637} C_VEL
LIN {X 0,Y 200.631,Z 654.624,A -85,B 0,C 180,E1 -21534.386,E2 -21534.386} C_VEL
LIN {X 0,Y 199.153,Z 659.758,A -85,B 0,C 180,E1 -21538.085,E2 -21538.085} C_VEL
LIN {X 0,Y 197.967,Z 664.078,A -85,B 0,C 180,E1 -21542.176,E2 -21542.176} C_VEL
LIN {X 0,Y 197.43,Z 666.358,A -85,B 0,C 180,E1 -21545.04,E2 -21545.04} C_VEL
LIN {X 0,Y 197.174,Z 668.169,A -85,B 0,C 180,E1 -21548.356,E2 -21548.356} C_VEL
LIN {X 0,Y 197.357,Z 669.423,A -85,B 0,C 180,E1 -21552.58,E2 -21552.58} C_VEL
LIN {X 0,Y 197.728,Z 669.581,A -85,B 0,C 180,E1 -21555.307,E2 -21555.307} C_VEL
LIN {X 0,Y 198.34,Z 669.243,A -85,B 0,C 180,E1 -21558.084,E2 -21558.084} C_VEL
LIN {X 0,Y 199.281,Z 668.378,A -85,B 0,C 180,E1 -21560.885,E2 -21560.885} C_VEL
LIN {X 0,Y 200.527,Z 666.882,A -85,B 0,C 180,E1 -21563.717,E2 -21563.717} C_VEL
LIN {X 0,Y 202.914,Z 663.793,A -85,B 0,C 180,E1 -21567.708,E2 -21567.708} C_VEL
LIN {X 0,Y 206.614,Z 658.677,A -85,B 0,C 180,E1 -21572.178,E2 -21572.178} C_VEL
LIN {X 0,Y 210.449,Z 653.203,A -85,B 0,C 180,E1 -21575.707,E2 -21575.707} C_VEL
LIN {X 0,Y 214.606,Z 646.861,A -85,B 0,C 180,E1 -21578.885,E2 -21578.885} C_VEL
LIN {X 0,Y 219.688,Z 638.806,A -85,B 0,C 180,E1 -21582.073,E2 -21582.073} C_VEL
LIN {X 0,Y 224.803,Z 629.879,A -85,B 0,C 180,E1 -21584.922,E2 -21584.922} C_VEL
LIN {X 0,Y 230.31,Z 619.504,A -85,B 0,C 180,E1 -21587.555,E2 -21587.555} C_VEL
LIN {X 0,Y 235.646,Z 608.381,A -85,B 0,C 180,E1 -21589.807,E2 -21589.807} C_VEL
LIN {X 0,Y 240.834,Z 596.292,A -85,B 0,C 180,E1 -21591.779,E2 -21591.779} C_VEL
LIN {X 0,Y 245.839,Z 582.591,A -85,B 0,C 180,E1 -21593.583,E2 -21593.583} C_VEL
LIN {X 0,Y 250.138,Z 568.661,A -85,B 0,C 180,E1 -21595.006,E2 -21595.006} C_VEL
LIN {X 0,Y 253.803,Z 553.719,A -85,B 0,C 180,E1 -21596.2,E2 -21596.2} C_VEL
LIN {X 0,Y 256.648,Z 538.632,A -85,B 0,C 180,E1 -21597.081,E2 -21597.081} C_VEL
LIN {X 0,Y 258.74,Z 522.499,A -85,B 0,C 180,E1 -21597.732,E2 -21597.732} C_VEL
LIN {X 0,Y 265.127,Z 455.967,A -85,B 0,C 180,E1 -21599.682,E2 -21599.682} C_VEL
LIN {X 0,Y 261.69,Z 448.831,A -85,B 0,C 180,E1 -21601.686,E2 -21601.686} C_VEL
LIN {X 0,Y 256.856,Z 439.802,A -85,B 0,C 180,E1 -21604.998,E2 -21604.998} C_VEL
LIN {X 0,Y 254.956,Z 436.769,A -85,B 0,C 180,E1 -21606.498,E2 -21606.498} C_VEL
LIN {X 0,Y 252.626,Z 433.085,A -85,B 0,C 180,E1 -21608.676,E2 -21608.676} C_VEL
LIN {X 0,Y 250.594,Z 430.021,A -85,B 0,C 180,E1 -21611.009,E2 -21611.009} C_VEL
LIN {X 0,Y 249.955,Z 428.94,A -85,B 0,C 180,E1 -21611.928,E2 -21611.928} C_VEL
LIN {X 0,Y 247.898,Z 426.438,A -85,B 0,C 180,E1 -21615.893,E2 -21615.893} C_VEL
LIN {X 0,Y 247.595,Z 425.007,A -85,B 0,C 180,E1 -21617.774,E2 -21617.774} C_VEL
LIN {X 0,Y 247.422,Z 425.736,A -85,B 0,C 180,E1 -21621.003,E2 -21621.003} C_VEL
LIN {X 0,Y 248.092,Z 427.18,A -85,B 0,C 180,E1 -21623.925,E2 -21623.925} C_VEL
LIN {X 0,Y 250.76,Z 433.032,A -85,B 0,C 180,E1 -21628.812,E2 -21628.812} C_VEL
LIN {X 0,Y 253.356,Z 438.304,A -85,B 0,C 180,E1 -21631.693,E2 -21631.693} C_VEL
LIN {X 0,Y 254.1,Z 440.264,A -85,B 0,C 180,E1 -21632.442,E2 -21632.442} C_VEL
LIN {X 0,Y 254.704,Z 442.809,A -85,B 0,C 180,E1 -21633.105,E2 -21633.105} C_VEL
LIN {X 0,Y 255.589,Z 448.857,A -85,B 0,C 180,E1 -21634.256,E2 -21634.256} C_VEL
LIN {X 0,Y 256.801,Z 456.744,A -85,B 0,C 180,E1 -21635.651,E2 -21635.651} C_VEL
LIN {X 0,Y 258.033,Z 460.702,A -85,B 0,C 180,E1 -21636.623,E2 -21636.623} C_VEL
LIN {X 0,Y 260.789,Z 468.831,A -85,B 0,C 180,E1 -21638.547,E2 -21638.547} C_VEL
LIN {X 0,Y 260.917,Z 469.281,A -85,B 0,C 180,E1 -21638.634,E2 -21638.634} C_VEL
LIN {X 0,Y 253.417,Z 542.78,A -85,B 0,C 180,E1 -21640.759,E2 -21640.759} C_VEL
LIN {X 0,Y 250.7,Z 558.534,A -85,B 0,C 180,E1 -21641.418,E2 -21641.418} C_VEL
LIN {X 0,Y 247.046,Z 573.771,A -85,B 0,C 180,E1 -21642.297,E2 -21642.297} C_VEL
LIN {X 0,Y 242.299,Z 589.39,A -85,B 0,C 180,E1 -21643.519,E2 -21643.519} C_VEL
LIN {X 0,Y 237.11,Z 603.475,A -85,B 0,C 180,E1 -21644.954,E2 -21644.954} C_VEL
LIN {X 0,Y 231.556,Z 616.698,A -85,B 0,C 180,E1 -21646.72,E2 -21646.72} C_VEL
LIN {X 0,Y 226.021,Z 628.311,A -85,B 0,C 180,E1 -21648.653,E2 -21648.653} C_VEL
LIN {X 0,Y 220.28,Z 639.284,A -85,B 0,C 180,E1 -21650.94,E2 -21650.94} C_VEL
LIN {X 0,Y 214.128,Z 650.158,A -85,B 0,C 180,E1 -21653.786,E2 -21653.786} C_VEL
LIN {X 0,Y 208.633,Z 659.283,A -85,B 0,C 180,E1 -21656.811,E2 -21656.811} C_VEL
LIN {X 0,Y 203.899,Z 666.933,A -85,B 0,C 180,E1 -21660.013,E2 -21660.013} C_VEL
LIN {X 0,Y 199.245,Z 674.219,A -85,B 0,C 180,E1 -21663.837,E2 -21663.837} C_VEL
LIN {X 0,Y 195.614,Z 680.074,A -85,B 0,C 180,E1 -21667.836,E2 -21667.836} C_VEL
LIN {X 0,Y 193.532,Z 683.643,A -85,B 0,C 180,E1 -21670.923,E2 -21670.923} C_VEL
LIN {X 0,Y 191.585,Z 687.264,A -85,B 0,C 180,E1 -21675.12,E2 -21675.12} C_VEL
LIN {X 0,Y 190.551,Z 689.732,A -85,B 0,C 180,E1 -21679.372,E2 -21679.372} C_VEL
LIN {X 0,Y 190.299,Z 691.068,A -85,B 0,C 180,E1 -21683.638,E2 -21683.638} C_VEL
LIN {X 0,Y 190.56,Z 691.259,A -85,B 0,C 180,E1 -21687.885,E2 -21687.885} C_VEL
LIN {X 0,Y 190.642,Z 690.876,A -85,B 0,C 180,E1 -21689.999,E2 -21689.999} C_VEL
LIN {X 0,Y 190.593,Z 690.167,A -85,B 0,C 180,E1 -21692.112,E2 -21692.112} C_VEL
LIN {X 0,Y 190.461,Z 688.749,A -85,B 0,C 180,E1 -21694.939,E2 -21694.939} C_VEL
LIN {X 0,Y 190.508,Z 685.159,A -85,B 0,C 180,E1 -21699.555,E2 -21699.555} C_VEL
LIN {X 0,Y 191.245,Z 680.417,A -85,B 0,C 180,E1 -21703.819,E2 -21703.819} C_VEL
LIN {X 0,Y 192.804,Z 674.209,A -85,B 0,C 180,E1 -21708.023,E2 -21708.023} C_VEL
LIN {X 0,Y 194.82,Z 667.304,A -85,B 0,C 180,E1 -21711.7,E2 -21711.7} C_VEL
LIN {X 0,Y 197.675,Z 659.026,A -85,B 0,C 180,E1 -21715.253,E2 -21715.253} C_VEL
LIN {X 0,Y 200.983,Z 649.007,A -85,B 0,C 180,E1 -21718.737,E2 -21718.737} C_VEL
LIN {X 0,Y 204.542,Z 638.762,A -85,B 0,C 180,E1 -21721.599,E2 -21721.599} C_VEL
LIN {X 0,Y 208.225,Z 627.662,A -85,B 0,C 180,E1 -21724.133,E2 -21724.133} C_VEL
LIN {X 0,Y 212.067,Z 615.746,A -85,B 0,C 180,E1 -21726.325,E2 -21726.325} C_VEL
LIN {X 0,Y 215.675,Z 602.865,A -85,B 0,C 180,E1 -21728.252,E2 -21728.252} C_VEL
LIN {X 0,Y 219.067,Z 588.87,A -85,B 0,C 180,E1 -21729.912,E2 -21729.912} C_VEL
LIN {X 0,Y 222.008,Z 574.629,A -85,B 0,C 180,E1 -21731.211,E2 -21731.211} C_VEL
LIN {X 0,Y 224.374,Z 560.392,A -85,B 0,C 180,E1 -21732.18,E2 -21732.18} C_VEL
LIN {X 0,Y 226.21,Z 545.448,A -85,B 0,C 180,E1 -21732.889,E2 -21732.889} C_VEL
LIN {X 0,Y 232.263,Z 456.875,A -85,B 0,C 180,E1 -21735.747,E2 -21735.747} C_VEL
LIN {X 0,Y 231.681,Z 453.626,A -85,B 0,C 180,E1 -21736.005,E2 -21736.005} C_VEL
LIN {X 0,Y 223.925,Z 434.915,A -85,B 0,C 180,E1 -21738.433,E2 -21738.433} C_VEL
LIN {X 0,Y 216.666,Z 419.242,A -85,B 0,C 180,E1 -21740.846,E2 -21740.846} C_VEL
LIN {X 0,Y 209.857,Z 405.97,A -85,B 0,C 180,E1 -21743.218,E2 -21743.218} C_VEL
LIN {X 0,Y 202.873,Z 393.384,A -85,B 0,C 180,E1 -21745.849,E2 -21745.849} C_VEL
LIN {X 0,Y 196.049,Z 382.271,A -85,B 0,C 180,E1 -21748.607,E2 -21748.607} C_VEL
LIN {X 0,Y 193.174,Z 378.069,A -85,B 0,C 180,E1 -21749.825,E2 -21749.825} C_VEL
LIN {X 0,Y 192.817,Z 377.036,A -85,B 0,C 180,E1 -21750.08,E2 -21750.08} C_VEL
LIN {X 0,Y 192.638,Z 376.113,A -85,B 0,C 180,E1 -21750.717,E2 -21750.717} C_VEL
LIN {X 0,Y 192.703,Z 376.106,A -85,B 0,C 180,E1 -21756.349,E2 -21756.349} C_VEL
LIN {X 0,Y 192.729,Z 376.096,A -85,B 0,C 180,E1 -21761.458,E2 -21761.458} C_VEL
LIN {X 0,Y 192.762,Z 376.097,A -85,B 0,C 180,E1 -21765.214,E2 -21765.214} C_VEL
LIN {X 0,Y 192.978,Z 376.026,A -85,B 0,C 180,E1 -21769.509,E2 -21769.509} C_VEL
LIN {X 0,Y 193.059,Z 376.038,A -85,B 0,C 180,E1 -21771.628,E2 -21771.628} C_VEL
LIN {X 0,Y 193.262,Z 376.011,A -85,B 0,C 180,E1 -21777.917,E2 -21777.917} C_VEL
LIN {X 0,Y 193.441,Z 375.995,A -85,B 0,C 180,E1 -21780.001,E2 -21780.001} C_VEL
LIN {X 0,Y 192.978,Z 376.067,A -85,B 0,C 180,E1 -21784.178,E2 -21784.178} C_VEL
LIN {X 0,Y 193.071,Z 376.036,A -85,B 0,C 180,E1 -21788.373,E2 -21788.373} C_VEL
LIN {X 0,Y 192.852,Z 376.086,A -85,B 0,C 180,E1 -21792.631,E2 -21792.631} C_VEL
LIN {X 0,Y 192.756,Z 376.069,A -85,B 0,C 180,E1 -21796.96,E2 -21796.96} C_VEL
LIN {X 0,Y 192.621,Z 376.115,A -85,B 0,C 180,E1 -21801.4,E2 -21801.4} C_VEL
LIN {X 0,Y 192.646,Z 376.09,A -85,B 0,C 180,E1 -21804.214,E2 -21804.214} C_VEL
LIN {X 0,Y 192.649,Z 376.106,A -85,B 0,C 180,E1 -21808.893,E2 -21808.893} C_VEL
LIN {X 0,Y 192.598,Z 376.101,A -85,B 0,C 180,E1 -21813.187,E2 -21813.187} C_VEL
LIN {X 0,Y 192.551,Z 376.122,A -85,B 0,C 180,E1 -21818.353,E2 -21818.353} C_VEL
LIN {X 0,Y 192.488,Z 376.106,A -85,B 0,C 180,E1 -21823.096,E2 -21823.096} C_VEL
LIN {X 0,Y 192.49,Z 376.133,A -85,B 0,C 180,E1 -21826.906,E2 -21826.906} C_VEL
LIN {X 0,Y 192.551,Z 376.103,A -85,B 0,C 180,E1 -21831.649,E2 -21831.649} C_VEL
LIN {X 0,Y 192.596,Z 376.109,A -85,B 0,C 180,E1 -21836.815,E2 -21836.815} C_VEL
LIN {X 0,Y 192.637,Z 376.115,A -85,B 0,C 180,E1 -21841.689,E2 -21841.689} C_VEL
LIN {X 0,Y 192.68,Z 376.106,A -85,B 0,C 180,E1 -21846.346,E2 -21846.346} C_VEL
LIN {X 0,Y 192.668,Z 376.23,A -85,B 0,C 180,E1 -21851.011,E2 -21851.011} C_VEL
LIN {X 0,Y 193.575,Z 378.779,A -85,B 0,C 180,E1 -21851.48,E2 -21851.48} C_VEL
LIN {X 0,Y 195.757,Z 381.097,A -85,B 0,C 180,E1 -21852.351,E2 -21852.351} C_VEL
LIN {X 0,Y 198.246,Z 384.959,A -85,B 0,C 180,E1 -21853.387,E2 -21853.387} C_VEL
LIN {X 0,Y 199.605,Z 386.733,A -85,B 0,C 180,E1 -21853.914,E2 -21853.914} C_VEL
LIN {X 0,Y 208.315,Z 399.187,A -85,B 0,C 180,E1 -21857.109,E2 -21857.109} C_VEL
LIN {X 0,Y 214.471,Z 409.111,A -85,B 0,C 180,E1 -21859.218,E2 -21859.218} C_VEL
LIN {X 0,Y 222.765,Z 422.943,A -85,B 0,C 180,E1 -21861.828,E2 -21861.828} C_VEL
LIN {X 0,Y 228.022,Z 433.266,A -85,B 0,C 180,E1 -21863.43,E2 -21863.43} C_VEL
LIN {X 0,Y 232.479,Z 442.146,A -85,B 0,C 180,E1 -21864.711,E2 -21864.711} C_VEL
LIN {X 0,Y 226.802,Z 524.888,A -85,B 0,C 180,E1 -21867.392,E2 -21867.392} C_VEL
LIN {X 0,Y 225.067,Z 540.359,A -85,B 0,C 180,E1 -21868.211,E2 -21868.211} C_VEL
LIN {X 0,Y 222.704,Z 555.77,A -85,B 0,C 180,E1 -21869.379,E2 -21869.379} C_VEL
LIN {X 0,Y 220.109,Z 569.034,A -85,B 0,C 180,E1 -21870.687,E2 -21870.687} C_VEL
LIN {X 0,Y 216.69,Z 583.772,A -85,B 0,C 180,E1 -21872.557,E2 -21872.557} C_VEL
LIN {X 0,Y 212.984,Z 597.351,A -85,B 0,C 180,E1 -21874.733,E2 -21874.733} C_VEL
LIN {X 0,Y 209.506,Z 608.775,A -85,B 0,C 180,E1 -21876.985,E2 -21876.985} C_VEL
LIN {X 0,Y 205.695,Z 620.478,A -85,B 0,C 180,E1 -21879.837,E2 -21879.837} C_VEL
LIN {X 0,Y 201.974,Z 631.039,A -85,B 0,C 180,E1 -21883.012,E2 -21883.012} C_VEL
LIN {X 0,Y 198.691,Z 640.235,A -85,B 0,C 180,E1 -21886.439,E2 -21886.439} C_VEL
LIN {X 0,Y 196.16,Z 647.475,A -85,B 0,C 180,E1 -21889.763,E2 -21889.763} C_VEL
LIN {X 0,Y 193.911,Z 654.069,A -85,B 0,C 180,E1 -21893.496,E2 -21893.496} C_VEL
LIN {X 0,Y 192.357,Z 659.238,A -85,B 0,C 180,E1 -21897.176,E2 -21897.176} C_VEL
LIN {X 0,Y 191.147,Z 663.428,A -85,B 0,C 180,E1 -21900.981,E2 -21900.981} C_VEL
LIN {X 0,Y 190.248,Z 667.065,A -85,B 0,C 180,E1 -21905.637,E2 -21905.637} C_VEL
LIN {X 0,Y 190.083,Z 668.79,A -85,B 0,C 180,E1 -21909.063,E2 -21909.063} C_VEL
LIN {X 0,Y 190.242,Z 669.778,A -85,B 0,C 180,E1 -21912.365,E2 -21912.365} C_VEL
LIN {X 0,Y 190.699,Z 670.019,A -85,B 0,C 180,E1 -21915.554,E2 -21915.554} C_VEL
LIN {X 0,Y 191.923,Z 669.252,A -85,B 0,C 180,E1 -21920.265,E2 -21920.265} C_VEL
LIN {X 0,Y 193.826,Z 667.315,A -85,B 0,C 180,E1 -21924.538,E2 -21924.538} C_VEL
LIN {X 0,Y 196.717,Z 663.868,A -85,B 0,C 180,E1 -21929.031,E2 -21929.031} C_VEL
LIN {X 0,Y 199.962,Z 659.721,A -85,B 0,C 180,E1 -21932.811,E2 -21932.811} C_VEL
LIN {X 0,Y 204.156,Z 654.12,A -85,B 0,C 180,E1 -21936.585,E2 -21936.585} C_VEL
LIN {X 0,Y 209.37,Z 646.738,A -85,B 0,C 180,E1 -21940.386,E2 -21940.386} C_VEL
LIN {X 0,Y 214.332,Z 639.243,A -85,B 0,C 180,E1 -21943.368,E2 -21943.368} C_VEL
LIN {X 0,Y 219.714,Z 630.291,A -85,B 0,C 180,E1 -21946.257,E2 -21946.257} C_VEL
LIN {X 0,Y 225.468,Z 620.004,A -85,B 0,C 180,E1 -21948.894,E2 -21948.894} C_VEL
LIN {X 0,Y 231.344,Z 608.361,A -85,B 0,C 180,E1 -21951.263,E2 -21951.263} C_VEL
LIN {X 0,Y 236.582,Z 596.588,A -85,B 0,C 180,E1 -21953.175,E2 -21953.175} C_VEL
LIN {X 0,Y 241.37,Z 584.071,A -85,B 0,C 180,E1 -21954.826,E2 -21954.826} C_VEL
LIN {X 0,Y 245.917,Z 570.079,A -85,B 0,C 180,E1 -21956.285,E2 -21956.285} C_VEL
LIN {X 0,Y 249.774,Z 555.374,A -85,B 0,C 180,E1 -21957.48,E2 -21957.48} C_VEL
LIN {X 0,Y 252.853,Z 540.005,A -85,B 0,C 180,E1 -21958.407,E2 -21958.407} C_VEL
LIN {X 0,Y 254.996,Z 524.824,A -85,B 0,C 180,E1 -21959.033,E2 -21959.033} C_VEL
LIN {X 0,Y 261.499,Z 459.492,A -85,B 0,C 180,E1 -21960.961,E2 -21960.961} C_VEL
LIN {X 0,Y 258.724,Z 453.685,A -85,B 0,C 180,E1 -21962.744,E2 -21962.744} C_VEL
LIN {X 0,Y 254.8,Z 445.927,A -85,B 0,C 180,E1 -21965.66,E2 -21965.66} C_VEL
LIN {X 0,Y 253.157,Z 443.257,A -85,B 0,C 180,E1 -21967.021,E2 -21967.021} C_VEL
LIN {X 0,Y 251.098,Z 439.778,A -85,B 0,C 180,E1 -21969.085,E2 -21969.085} C_VEL
LIN {X 0,Y 249.123,Z 436.573,A -85,B 0,C 180,E1 -21971.534,E2 -21971.534} C_VEL
LIN {X 0,Y 248.568,Z 435.777,A -85,B 0,C 180,E1 -21972.345,E2 -21972.345} C_VEL
LIN {X 0,Y 246.67,Z 433.037,A -85,B 0,C 180,E1 -21976.553,E2 -21976.553} C_VEL
LIN {X 0,Y 246.522,Z 432.024,A -85,B 0,C 180,E1 -21977.854,E2 -21977.854} C_VEL
LIN {X 0,Y 246.37,Z 432.811,A -85,B 0,C 180,E1 -21981.097,E2 -21981.097} C_VEL
LIN {X 0,Y 246.91,Z 434.012,A -85,B 0,C 180,E1 -21983.595,E2 -21983.595} C_VEL
LIN {X 0,Y 249.262,Z 439.587,A -85,B 0,C 180,E1 -21988.288,E2 -21988.288} C_VEL
LIN {X 0,Y 251.874,Z 445.465,A -85,B 0,C 180,E1 -21991.414,E2 -21991.414} C_VEL
LIN {X 0,Y 254.437,Z 451.457,A -85,B 0,C 180,E1 -21993.805,E2 -21993.805} C_VEL
LIN {X 0,Y 257.103,Z 458.252,A -85,B 0,C 180,E1 -21995.945,E2 -21995.945} C_VEL
LIN {X 0,Y 258.033,Z 460.702,A -85,B 0,C 180,E1 -21996.623,E2 -21996.623} C_VEL
LIN {X 0,Y 258.711,Z 463.433,A -85,B 0,C 180,E1 -21997.178,E2 -21997.178} C_VEL
